# B&R Automation Studio project vibratorControlWithCurrentController (part 3)

#### brdkEM.c - Represents an equipment module.
```c
#include <brdkEM_func.h>

void brdkEM(struct brdkEM* this) {

	brdkEM_typ* parent;
	wakeMU(this->internal.muList.idx,(unsigned long)this);
	parent = getEm(this->internal.muList.parentIdx);

	/* if enabled command state completet can be set by settings the sub state to SC (65000) */
	if(this->setup.useSubstateSC) this->internal.cmdSC = this->substate == SC ? true : this->cmd.sc;
	else this->internal.cmdSC = this->cmd.sc;

	/* update information about the last */

	switch(this->state) {

		case STATE_STOPPED:
			this->status.color = BLUE;
			lightTree(this,BLUE,RED);
			setSubStateText(this);
			observeChildrensState(this, 2, STATE_ABORTING, STATE_ABORTED);						/* check if a child is in STATE- ABORTING or ABORTED */
			observeParentState(this, parent, 2, STATE_RESETTING, STATE_ABORTING);					/* check if parent is in STATE- RESETTING */
			if(this->internal.findParent) findParent(this,parent,STATE_RESETTING,11,STATE_IDLE,STATE_STARTING,STATE_EXECUTE,STATE_HOLDING,STATE_HELD,STATE_UNHOLDING,STATE_SUSPENDING,STATE_SUSPENDED,STATE_UNSUSPENDING,STATE_COMPLETING,STATE_COMPLETE);
			checkCommands(this, parent, 3, STATE_RESETTING, STATE_ABORTING, STATE_DEACTIVATING);		/* check commands reset, abort, not activate */
			setChildrenMode(this);
			if(this->mode == MODE_UNDEFINED) this->mode = MODE_PRODUCING;
			this->status.level = parent != NULL ? parent->status.level+1  : 0;	/* sets the hierarchy level */
			break;

		case STATE_RESETTING:
			this->status.color = WHITE;
			lightTree(this,BLUE,WHITE);
			setSubStateText(this);
			checkChildren(this, STATE_IDLE); 													/* CHECK IF ALL CHILDREN ARE IN STATE_IDLE */
			observeChildrensState(this, 3, STATE_ABORTING, STATE_ABORTED, STATE_STOPPING);		/* CHECK IF ONE CHILD IS IN STATE_ABORTING OR STATE_ABORTED */
			observeParentState(this,parent, 2, STATE_STOPPING,STATE_ABORTING);							/* checks if parent is in STATE- STOPPING or ABORTING */
			checkCommands(this, parent, 2, STATE_STOPPING, STATE_ABORTING);								/* check commands stop and abort */
			break;

		case STATE_IDLE:
			this->status.color = BLUE;
			lightTree(this,BLUE,WHITE);
			setSubStateText(this);
			observeChildrensState(this, 4, STATE_ABORTING, STATE_ABORTED, STATE_STOPPING, STATE_STOPPED);		/* check child state */
			observeParentState(this, parent, 3,STATE_STARTING,STATE_STOPPING,STATE_ABORTING);						/* CHECK STATE OF THE PARENT AND MAYBE FOLLOW */
			if(this->internal.findParent) findParent(this,parent,STATE_STARTING,9,STATE_EXECUTE,STATE_HOLDING,STATE_HELD,STATE_UNHOLDING,STATE_SUSPENDING,STATE_SUSPENDED,STATE_UNSUSPENDING,STATE_COMPLETING,STATE_COMPLETE);
			checkCommands(this, parent, 3, STATE_STOPPING, STATE_ABORTING, STATE_STARTING);								/* check commands stop, abort, start */
			break;

		case STATE_STARTING:
			this->status.color = WHITE;
			lightTree(this,flashColor(this,GREEN),WHITE);
			setSubStateText(this);
			checkChildren(this, STATE_EXECUTE); 															/* SUBSTATE MUST BE IN SC - CHECK IF ALL CHILDREN ARE IN STATE_EXECUTE */
			observeChildrensState(this, 4, STATE_ABORTING, STATE_ABORTED, STATE_STOPPING, STATE_STOPPED);	/* CHECK IF ONE CHILD IS IN STATE */
			observeParentState(this, parent,2,STATE_STOPPING,STATE_ABORTING); 										/* CHECK STATE OF THE PARENT AND MAYBE FOLLOW */
			checkCommands(this, parent, 2, STATE_STOPPING, STATE_ABORTING);											/* check commands stop, abort */
			break;

		case STATE_EXECUTE:
			this->status.color = GREEN;
			lightTree(this,GREEN,WHITE);
			setSubStateText(this);
			observeChildrensState(this, 8, STATE_ABORTING, STATE_ABORTED, STATE_STOPPING, STATE_STOPPED, STATE_SUSPENDING, STATE_SUSPENDED, STATE_HOLDING, STATE_HELD);		/* CHECK IF ONE CHILD IS IN STATE */
			observeParentState(this,parent,5,STATE_HOLDING,STATE_SUSPENDING,STATE_COMPLETING,STATE_STOPPING,STATE_ABORTING); /* CHECK STATE OF THE PARENT AND MAYBE FOLLOW */
			if(this->internal.findParent) findParent(this,parent,STATE_EXECUTE,7,STATE_HOLDING,STATE_HELD,STATE_SUSPENDING,STATE_SUSPENDED,STATE_COMPLETING,STATE_COMPLETE);
			checkCommands(this, parent, 5, STATE_STOPPING, STATE_ABORTING, STATE_HOLDING, STATE_SUSPENDING, STATE_COMPLETING);		/* check commands stop, abort, hold, suspend, complete */
			break;

		case STATE_HOLDING:
			this->status.color = WHITE;
			lightTree(this,flashColor(this,RED),WHITE);
			setSubStateText(this);
			checkChildren(this, STATE_HELD); 											/* SUBSTATE MUST BE IN SC - CHECK IF ALL CHILDREN ARE IN STATE_EXECUTE */
			observeChildrensState(this, 2, STATE_ABORTING, STATE_ABORTED);				/* CHECK IF ONE CHILD IS IN STATE */
			observeParentState(this,parent,2,STATE_STOPPING,STATE_ABORTING); 					/* CHECK STATE OF THE PARENT AND MAYBE FOLLOW */
			checkCommands(this, parent, 2, STATE_STOPPING, STATE_ABORTING);						/* check commands stop, abort */
			break;

		case STATE_HELD:
			this->status.color = RED;
			lightTree(this,flashColor(this,RED),WHITE);
			setSubStateText(this);
			observeChildrensState(this, 2, STATE_ABORTING, STATE_ABORTED);					/* CHECK IF ONE CHILD IS IN STATE */
			observeParentState(this,parent,3,STATE_UNHOLDING,STATE_STOPPING,STATE_ABORTING); 	/* CHECK STATE OF THE PARENT AND MAYBE FOLLOW */
			if(this->internal.findParent) findParent(this,parent,STATE_UNHOLDING,6,STATE_EXECUTE,STATE_SUSPENDING,STATE_SUSPENDED,STATE_UNSUSPENDING,STATE_COMPLETING,STATE_COMPLETE);
			checkCommands(this, parent, 3, STATE_STOPPING, STATE_ABORTING, STATE_UNHOLDING);		/* check commands stop, abort, start */
			break;

		case STATE_UNHOLDING:
			this->status.color = WHITE;
			lightTree(this,RED,GREEN);
			setSubStateText(this);
			checkChildren(this, STATE_EXECUTE); 											/* SUBSTATE MUST BE IN SC - CHECK IF ALL CHILDREN ARE IN STATE_EXECUTE */
			observeChildrensState(this, 2, STATE_ABORTING, STATE_ABORTED);					/* CHECK IF ONE CHILD IS IN STATE */
			observeParentState(this,parent,2,STATE_STOPPING,STATE_ABORTING); 						/* CHECK STATE OF THE PARENT AND MAYBE FOLLOW */
			checkCommands(this, parent, 2, STATE_STOPPING, STATE_ABORTING);							/* check commands stop, abort */
			break;

		case STATE_SUSPENDING:
			this->status.color = WHITE;
			lightTree(this,ORANGE,WHITE);
			setSubStateText(this);
			checkChildren(this, STATE_SUSPENDED); 											/* SUBSTATE MUST BE IN SC - CHECK IF ALL CHILDREN ARE IN STATE_EXECUTE */
			observeChildrensState(this, 2, STATE_ABORTING, STATE_ABORTED);					/* CHECK IF ONE CHILD IS IN STATE */
			observeParentState(this,parent,2,STATE_STOPPING,STATE_ABORTING); 						/* CHECK STATE OF THE PARENT AND MAYBE FOLLOW */
			checkCommands(this, parent, 2, STATE_STOPPING, STATE_ABORTING);							/* check commands stop, abort */
			break;

		case STATE_SUSPENDED:
			this->status.color = ORANGE;
			lightTree(this,ORANGE,WHITE);
			setSubStateText(this);
			observeChildrensState(this, 2, STATE_ABORTING, STATE_ABORTED);					/* CHECK IF ONE CHILD IS IN STATE */
			observeParentState(this,parent,3,STATE_UNSUSPENDING,STATE_STOPPING,STATE_ABORTING); 	/* CHECK STATE OF THE PARENT AND MAYBE FOLLOW */
			if(this->internal.findParent) findParent(this,parent,STATE_UNSUSPENDING,6,STATE_EXECUTE,STATE_HOLDING,STATE_HELD,STATE_UNHOLDING,STATE_COMPLETING,STATE_COMPLETE);
			checkCommands(this, parent, 3, STATE_STOPPING, STATE_ABORTING, STATE_UNSUSPENDING);		/* check commands stop, abort, start */
			break;

		case STATE_UNSUSPENDING:
			this->status.color = WHITE;
			lightTree(this,ORANGE,GREEN);
			setSubStateText(this);
			checkChildren(this, STATE_EXECUTE); 											/* SUBSTATE MUST BE IN SC - CHECK IF ALL CHILDREN ARE IN STATE_EXECUTE */
			observeChildrensState(this, 2, STATE_ABORTING, STATE_ABORTED);					/* CHECK IF ONE CHILD IS IN STATE */
			observeParentState(this,parent,2,STATE_STOPPING,STATE_ABORTING); 						/* CHECK STATE OF THE PARENT AND MAYBE FOLLOW */
			checkCommands(this, parent, 2, STATE_STOPPING, STATE_ABORTING);							/* check commands stop, abort */
			break;

		case STATE_COMPLETING:
			this->status.color = WHITE;
			lightTree(this,GREEN,BLUE);
			setSubStateText(this);
			checkChildren(this, STATE_COMPLETE); 											/* SUBSTATE MUST BE IN SC - CHECK IF ALL CHILDREN ARE IN STATE_EXECUTE */
			observeChildrensState(this, 2, STATE_ABORTING, STATE_ABORTED);					/* CHECK IF ONE CHILD IS IN STATE */
			observeParentState(this,parent,2,STATE_STOPPING,STATE_ABORTING); 						/* CHECK STATE OF THE PARENT AND MAYBE FOLLOW */
			checkCommands(this, parent, 2, STATE_STOPPING, STATE_ABORTING);							/* check commands stop, abort */
			break;

		case STATE_COMPLETE:
			this->status.color = BLUE;
			lightTree(this,flashColor(this,BLUE),WHITE);
			setSubStateText(this);
			observeChildrensState(this, 2, STATE_ABORTING, STATE_ABORTED);					/* CHECK IF ONE CHILD IS IN STATE */
			observeParentState(this,parent,3,STATE_RESETTING,STATE_STOPPING,STATE_ABORTING); 		/* CHECK STATE OF THE PARENT AND MAYBE FOLLOW */
			if(this->internal.findParent) findParent(this,parent,STATE_RESETTING,10,STATE_IDLE,STATE_STARTING,STATE_EXECUTE,STATE_HOLDING,STATE_HELD,STATE_UNHOLDING,STATE_SUSPENDING,STATE_SUSPENDED,STATE_UNSUSPENDING,STATE_COMPLETING);
			checkCommands(this, parent, 3, STATE_STOPPING, STATE_ABORTING, STATE_RESETTING);		/* check commands stop, abort, reset */
			break;

		case STATE_ABORTING:
			this->status.color = WHITE;
			lightTree(this,RED,WHITE);
			setSubStateText(this);
			checkChildren(this, STATE_ABORTED);
			break;

		case STATE_ABORTED:
			this->status.color = RED;
			lightTree(this,RED,WHITE);
			setSubStateText(this);
			observeParentState(this,parent,1,STATE_CLEARING); 										/* CHECK STATE OF THE PARENT AND MAYBE FOLLOW */
			checkCommands(this, parent, 2, STATE_CLEARING, STATE_DEACTIVATING);						/* check commands clar, not activate */
			break;

		case STATE_CLEARING:
			this->status.color = WHITE;
			lightTree(this,RED,flashColor(this,BLUE));
			setSubStateText(this);
			checkChildren(this, STATE_STOPPED); 										/* SUBSTATE MUST BE IN SC - CHECK IF ALL CHILDREN ARE IN STATE_EXECUTE */
			observeChildrensState(this, 2, STATE_ABORTING, STATE_ABORTED);				/* CHECK IF ONE CHILD IS IN STATE */
			observeParentState(this,parent,2,STATE_STOPPING,STATE_ABORTING); 			/* CHECK STATE OF THE PARENT AND MAYBE FOLLOW */
			break;

		case STATE_STOPPING:
			this->status.color = WHITE;
			lightTree(this,GREEN,BLUE);
			setSubStateText(this);
			checkChildren(this, STATE_STOPPED); 									/* SUBSTATE MUST BE IN SC - CHECK IF ALL CHILDREN ARE IN STATE_EXECUTE */
			observeChildrensState(this, 2, STATE_ABORTING, STATE_ABORTED);			/* CHECK IF ONE CHILD IS IN STATE */
			observeParentState(this,parent,1,STATE_ABORTING); 								/* CHECK STATE OF THE PARENT AND MAYBE FOLLOW */
			checkCommands(this, parent, 2, STATE_ABORTING, STATE_DEACTIVATING);								/* check commands abort */
			break;

		case STATE_DEACTIVATING:
			this->status.color = WHITE;
			lightTree(this,flashColor(this,GREY),WHITE);
			setSubStateText(this);
			this->mode = MODE_UNDEFINED;
			this->internal.initSubstate = 0;
			if(this->internal.cmdSC) {
				UnregisterChild(this, parent);
				this->state = STATE_DEACTIVATED;
			}
			break;

		case STATE_ACTIVATING:
			this->status.color = WHITE;
			lightTree(this,flashColor(this,GREY),BLUE);
			setSubStateText(this);
			if(this->internal.cmdSC) {
				if(parent != NULL) {
					switch(parent->state) {

						case STATE_STOPPED:
							if(this->mode == MODE_UNDEFINED && this->setup.reactTo == BRDK_EM_REACT_TO_NONE) this->mode = MODE_PRODUCING;
							else this->mode = parent->mode;
							this->state = STATE_STOPPED;
							break;

						case STATE_DEACTIVATED:
							brdkStrCpy((unsigned long)this->status.substate,(unsigned long)"waiting for parent to be activated");
							break;

						default:
							brdkStrCpy((unsigned long)this->status.substate,(unsigned long)"waiting for parent to be in STATE_STOPPED");
							break;

					}
				}
				else {
					if(this->mode == MODE_UNDEFINED) this->mode = MODE_PRODUCING;
					this->state = STATE_STOPPED;
				}
			}
			break;

		case STATE_DEACTIVATED:
			brdkStrCpy((unsigned long)this->status.state,(unsigned long)brdkEMStateToA(this->state));
			this->status.color = GREY;
			lightTree(this,GREY,WHITE);
			setSubStateText(this);
			if(this->status.mode[0] == 0) brdkStrCpy((unsigned long)this->status.mode,brdkEMModeToA(this->mode));
			if(this->status.cycleTime == 0) this->status.cycleTime = getCycleTime();								/* get the modules cycle time */
			brdkEMInitialize(this,parent);
			checkCommands(this, parent, 1, STATE_ACTIVATING);
			break;
	}

	/* mode change */
	if(this->mode != this->internal.old.mode) {
		if(this->state == STATE_STOPPED || this->state == STATE_ACTIVATING || this->state == STATE_DEACTIVATING || this->state == STATE_DEACTIVATED) {
			/* save last state for log */
			if(this->setup.lastActivated) {
				brdkStrMemMove((unsigned long)this->status.last[1],(unsigned long)this->status.last[0], sizeof(this->status.last[0])*BRDK_MU_MAX_LAST_SIZE);
				brdkStrCpy((unsigned long)this->status.last[0], brdkEMModeToA(this->internal.old.mode));
				brdkStrCat((unsigned long)this->status.last[0], (unsigned long)"-->");
				brdkStrCat((unsigned long)this->status.last[0], brdkEMModeToA(this->mode));
			}
			this->internal.old.mode = this->mode;
			brdkStrCpy((unsigned long)this->status.mode,brdkEMModeToA(this->mode));
		}
		else { /* avoid mode being change in other states than STATE_STOPPED */
			this->status.unvalidatedMode = true;
			this->mode = this->internal.old.mode;
		}
	}

	this->status.time += this->status.cycleTime/1000;

	/* state change */
	if(this->state != this->internal.old.state || this->substate != this->internal.old.substate) {
		/* save last state for log */
		if(this->setup.lastActivated) {
			brdkStrMemMove((unsigned long)this->status.last[1],(unsigned long)this->status.last[0], sizeof(this->status.last[0])*BRDK_MU_MAX_LAST_SIZE);
			brdkStrCpy((unsigned long)this->status.last[0],(unsigned long)this->status.state);
			brdkStrCat((unsigned long)this->status.last[0],(unsigned long)": ");
			if(this->state != this->internal.old.state) brdkStrAppendUdintToA(this->substate,(unsigned long)this->status.last[0],BRDK_STR_CONVERT_DECIMAL,-1);
			else brdkStrAppendUdintToA(this->internal.old.substate,(unsigned long)this->status.last[0],BRDK_STR_CONVERT_DECIMAL,-1);
			brdkStrCat((unsigned long)this->status.last[0],(unsigned long)": ");
			brdkStrAppendUdintToA(this->status.time,(unsigned long)this->status.last[0],BRDK_STR_CONVERT_DECIMAL,-1);
			brdkStrCat((unsigned long)this->status.last[0],(unsigned long)"ms");
		}
		brdkStrCpy((unsigned long)this->status.state,(unsigned long)brdkEMStateToA(this->state));
		if(this->state != this->internal.old.state) {
			/* log who interrupted the module */
			if(this->internal.pInterrupter != 0 && this->status.interruptedBy.name[0] == 0) {
				brdkStrCpy((unsigned long)this->status.interruptedBy.name,(unsigned long)((brdkEM_typ*)this->internal.pInterrupter)->status.name);
				if(this->internal.pInterrupter != (unsigned long)this) {
					this->status.interruptedBy.state = ((brdkEM_typ*)this->internal.pInterrupter)->status.interruptedBy.state;
					this->status.interruptedBy.substate = ((brdkEM_typ*)this->internal.pInterrupter)->status.interruptedBy.substate;
				}
				else {
					this->status.interruptedBy.state = ((brdkEM_typ*)this->internal.pInterrupter)->internal.old.state;
					this->status.interruptedBy.substate = ((brdkEM_typ*)this->internal.pInterrupter)->internal.old.substate;
				}
				if(this->state == STATE_ABORTING || this->state == STATE_STOPPING) {
					if(this->setup.lastActivated) {
						brdkStrMemMove((unsigned long)this->status.last[1],(unsigned long)this->status.last[0], sizeof(this->status.last[0])*BRDK_MU_MAX_LAST_SIZE);
						if(this->state == STATE_ABORTING) brdkStrCpy((unsigned long)this->status.last[0],(unsigned long)"Aborted by: ");
						else brdkStrCpy((unsigned long)this->status.last[0],(unsigned long)"Stopped by: ");
						brdkStrCat((unsigned long)this->status.last[0],(unsigned long)this->status.interruptedBy.name);
						brdkStrCat((unsigned long)this->status.last[0],(unsigned long)": ");
						brdkStrCat((unsigned long)this->status.last[0],brdkEMStateToA(this->status.interruptedBy.state));
						brdkStrCat((unsigned long)this->status.last[0],(unsigned long)": ");
						brdkStrAppendUdintToA(this->status.interruptedBy.substate,(unsigned long)this->status.last[0],BRDK_STR_CONVERT_DECIMAL,-1);
					}
				}
			}
			this->internal.cmdSC = this->cmd.sc = this->cmd.start = this->cmd.reset = this->cmd.abort = this->cmd.stop = this->cmd.clear = this->cmd.hold = this->cmd.complete = this->cmd.suspend = false; /* reset commands when the state changes */
			this->substate = 0;	/* reset substate by a state change */
			this->status.time = 0;
			this->status.unvalidatedMode = false;
		}
		this->status.substate[0] = this->description[0] = 0;
		this->internal.old.state = this->state;
		this->internal.old.substate = this->substate;

	}

	/* update parent info */
	if(parent != NULL) {
		this->status.parent.state = parent->state;
		this->status.parent.substate = parent->substate;
		this->status.parent.sleeping = parent->status.sleeping;
		this->status.parent.mode = parent->mode;
		this->status.parent.sc = parent->cmd.sc;
		if(parent->setup.skipStopSC) this->setup.skipStopSC = true; /* check if skipStopSC is set in parent module */
	}

	/* reactTo has changed */
	if(this->internal.old.reactTo != this->setup.reactTo) {
		if(this->setup.reactTo == BRDK_EM_REACT_TO_ALL) {
			if(parent != NULL) this->internal.findParent = true;
		}
		this->internal.old.reactTo = this->setup.reactTo;
	}

	/* update siblings info */
	updateSiblingInfo(&this->internal.muList.siblingIdx, &this->status.sibling[0]);

	/* save the restore information */
	if(this->setup.restore.activate) {
		if(this->setup.restore.pRestoreStruct != 0) {
			this->setup.restore.pRestoreStruct->mode = this->mode;
			this->setup.restore.pRestoreStruct->state = this->state;
			this->setup.restore.pRestoreStruct->substate = this->substate;
			this->setup.restore.pRestoreStruct->sc = this->internal.cmdSC;
		}
	}
}
```

#### brdkEMSleep.c - Put an equipment module to sleep. It's pointer is added to a sleeping module list where it can be found again by brdkEMWake().
```c
#include <brdkMU_func.h>

signed long brdkEMSleep(unsigned long pEM) {
	brdkEM_typ* this;
	if(pEM != 0) {
		this = (brdkEM_typ*)pEM;
		this->status.sleeping = true;
		if(this->setup.lastActivated) {
			brdkStrMemMove((unsigned long)this->status.last[1],(unsigned long)this->status.last[0], sizeof(this->status.last[0])*BRDK_MU_MAX_LAST_SIZE);
			brdkStrCpy((unsigned long)this->status.last[0],(unsigned long)"module put to sleep");
		}
		return sleepMU(this->internal.muList.idx, pEM);
	}
	return -1;
}
```

#### brdkEMModeToA.c - Converts an equipment module mode constant to a string representation.
```c
#include <brdkEM_func.h>

unsigned long brdkEMModeToA(signed long mode) {
	unsigned long pStr;
	switch(mode) {
		case MODE_UNDEFINED: 	pStr = (unsigned long)&"MODE_UNDEFINED"; 	break;	/* 0 */
		case MODE_PRODUCING: 	pStr = (unsigned long)&"MODE_PRODUCING"; 	break;	/* 1 */
		case MODE_MAINTENANCE: 	pStr = (unsigned long)&"MODE_MAINTENANCE"; 	break;	/* 2 */
		case MODE_MANUAL: 		pStr = (unsigned long)&"MODE_MANUAL"; 		break;	/* 3 */
		case MODE_CLEAN: 		pStr = (unsigned long)&"MODE_CLEAN"; 		break;	/* 16 */
		case MODE_JOG: 			pStr = (unsigned long)&"MODE_JOG"; 			break;	/* 17 */
		case MODE_CIP: 			pStr = (unsigned long)&"MODE_CIP"; 			break;	/* 18 */
		case MODE_CALIBRATING: 	pStr = (unsigned long)&"MODE_CALIBRATING"; 	break;	/* 19 */
		default: pStr = (unsigned long)&""; 	break;
	}
	return pStr;
}
```

#### brdkEM_func.c - Internal functions for brdkEM.
```c
#include <brdkEM_func.h>

static unsigned char semCreator = false;
SemCreate_typ SemCreateMUList;

/* initialize the equipment module */
void brdkEMInitialize(brdkEM_typ* this, brdkEM_typ* parent) {
	int i;
	brdk_mu_setup_module_typ module;

	switch(this->internal.initSubstate) {

		case 0:
			if(this->setup.name[0] == 0) ST_name(0,(char*)&this->setup.name,(unsigned char)0); 														/* set module name to task name if not set*/
			brdkStrCpy((unsigned long)this->status.name,(unsigned long)this->setup.name);
			if(this->setup.nameIdx > -1) brdkStrAppendUdintToA(this->setup.nameIdx,(unsigned long)&this->status.name, BRDK_STR_CONVERT_DECIMAL,-1);	/* add index to task name */
			this->internal.muList.parentIdx = -1;
			for(i=0; i<= BRDK_EM_MAX_CHILDREN; i++) this->internal.muList.childrenIdx[i] = -1;
			for(i=0; i<= BRDK_MU_MAX_SIBLINGS; i++) this->internal.muList.siblingIdx[i] = -1;
			if(!semCreator) {
				brdkStrCpy((unsigned long)this->status.substate,(unsigned long)"creating global semaphore");
				semCreator = true;
				this->internal.initSubstate = 10;
			}
			else this->internal.initSubstate = 20;
			break;

		case 10:
			SemCreateMUList.enable = true;
			SemCreateMUList.initCount = 0;
			SemCreateMUList.maxCount = 1;
			SemCreate(&SemCreateMUList);
			if(SemCreateMUList.status != ERR_OK) brdkStrCpy((unsigned long)this->status.substate,(unsigned long)"creating global semaphore");
			else {
				SemRelease(SemCreateMUList.ident);
				this->internal.muList.idx = addToMUList((unsigned long)this,0);
				if(this->internal.muList.idx != -1) {
					emListReady = true;
					this->internal.initSubstate = !this->setup.parent.name[0] ? 40 : 30;	/* check if the module has a parent name assigned */
				}
				else {
					brdkStrCpy((unsigned long)this->status.substate,(unsigned long)"em list full. Expand BRDK_EM_MAX_EMS.");
					this->internal.initSubstate = 200;
				}
			}
			break;

		case 20:	/* add module to em list */
			if(!emListReady) brdkStrCpy((unsigned long)this->status.substate,(unsigned long)"waiting for em list to be ready");
			else {
				brdkStrCpy((unsigned long)module.name,(unsigned long)this->setup.name);
				module.index = this->setup.nameIdx;
				this->internal.muList.idx = getMUIndex((unsigned long)this, &module);
				if(this->internal.muList.idx != -1) {
					if(moduleSleeping(this->internal.muList.idx)) {
						wakeMU(this->internal.muList.idx,(unsigned long)this);
						if(this->setup.lastActivated) {
							brdkStrMemMove((unsigned long)this->status.last[1],(unsigned long)this->status.last[0], sizeof(this->status.last[0])*BRDK_MU_MAX_LAST_SIZE);
							brdkStrCpy((unsigned long)this->status.last[0],(unsigned long)"module awake");
						}
						this->internal.initSubstate = 65000;
					}
					else {	/* module name already exists in the list */
						brdkStrCpy((unsigned long)this->status.substate,(unsigned long)"module name ");
						brdkStrCat((unsigned long)this->status.substate,(unsigned long)module.name);
						brdkStrCat((unsigned long)this->status.substate,(unsigned long)" already used. Rename module.");
						this->internal.muList.idx = -1;
						this->internal.initSubstate = 100;
					}
				}
				else {
					if(SemAcquire(SemCreateMUList.ident) != ERR_OK) brdkStrCpy((unsigned long)this->status.substate,(unsigned long)"waiting global semaphore to be free");
					else {
						this->internal.muList.idx = addToMUList((unsigned long)this,0);
						SemRelease(SemCreateMUList.ident);
						brdkStrCpy((unsigned long)this->status.substate,(unsigned long)"module added em list");
						if(this->internal.muList.idx != -1) this->internal.initSubstate = !this->setup.parent.name[0] ? 40 : 30;	/* check if the module has a parent name assigned */
						else {
							brdkStrCpy((unsigned long)this->status.substate,(unsigned long)"em list full. Expand BRDK_EM_MAX_EMS.");
							this->internal.initSubstate = 200;
						}
					}
				}
			}
			break;

		case 30:	/* find parent */
			this->internal.muList.parentIdx = getMUIndex((unsigned long)this, &this->setup.parent);
			if(this->internal.muList.parentIdx == -1) brdkStrCpy((unsigned long)this->status.substate,(unsigned long)"parent not found");
			else this->internal.initSubstate = 40;
			break;

		case 40:	/* find siblings */
			for(i=0; i<= BRDK_MU_MAX_SIBLINGS; i++) {
				if(this->setup.sibling[i].name[0] != 0) {
					this->internal.muList.siblingIdx[i] = getMUIndex((unsigned long)this, &this->setup.sibling[i]);
					if(this->internal.muList.siblingIdx[i] == -1) {
						brdkStrCpy((unsigned long)this->status.substate,(unsigned long)"sibling: ");
						brdkStrCat((unsigned long)this->status.substate,(unsigned long)this->setup.sibling[i].name);
						brdkStrCat((unsigned long)this->status.substate,(unsigned long)" not found");
						break;
					}
				}
			}
			if(i>=BRDK_MU_MAX_SIBLINGS) {
				this->status.substate[0] = 0;	/* reset status text */
				this->internal.initSubstate = this->internal.SemCreate_0.ident == 0 ? 50 : 60;
			}
			break;

		case 50:
			this->internal.SemCreate_0.enable = true;
			this->internal.SemCreate_0.initCount = 0;
			this->internal.SemCreate_0.maxCount = 1;
			SemCreate(&this->internal.SemCreate_0);
			switch(this->internal.SemCreate_0.status) {

				case 0:	/* ERR_OK */
					SemRelease(this->internal.SemCreate_0.ident);		/* release the semaphore so it's ready */
					this->internal.initSubstate = 60;
					break;

				case 65535:	/* ERR_FUB_BUSY */
					break;

				default:
					brdkStrCpy((unsigned long)this->status.substate,(unsigned long)"error creating the semaphore");
					break;

			}
			break;

		case 60:
			brdkStrCpy((unsigned long)this->status.substate,(unsigned long)"register child to parent");
			if(RegisterChild(this, parent) == 0) {
				this->internal.initSubstate = 65000;				/* add child to parent's children list */
				if(this->substate == 0) this->substate = 65000;		/* if substate is still 0 it's auto set to SC */
			}
			break;

		case 100: /* error module name already used. Check if anme is being changed */
			if(brdkStrCmp((unsigned long)module.name,(unsigned long)this->setup.name) != 0) {
				this->internal.initSubstate = 20;
			}
			break;

	}
}

/* traverse and find the real interrupter */
unsigned long findInterrupter(unsigned long pEM) {
	if(((brdkEM_typ*)pEM)->internal.pInterrupter != pEM) return findInterrupter(((brdkEM_typ*)pEM)->internal.pInterrupter);
	return pEM;
}

/* flash functionality */
brdk_em_color_typ flashColor(brdkEM_typ* this, brdk_em_color_typ color) {
	if(this->internal.flashTime >= BRDK_EM_FLASH_TIME*2) this->internal.flashTime = 0;
	else this->internal.flashTime += this->status.cycleTime/1000;
	return this->internal.flashTime >= BRDK_EM_FLASH_TIME ? color : WHITE;
}

/* light tree functionality */
void lightTree(brdkEM_typ* this, brdk_em_color_typ color1, brdk_em_color_typ color2) {
	this->status.lightTree.red 		= color1 == RED || color2 == RED;
	this->status.lightTree.yellow 	= color1 == ORANGE || color2 == ORANGE;
	this->status.lightTree.blue 	= color1 == BLUE || color2 == BLUE;
	this->status.lightTree.green 	= color1 == GREEN || color2 == GREEN;
}

/* set default sub state text if not set in program */
void setSubStateText(brdkEM_typ* this) {
	if(this->status.substate[0] == 0) {
		if(this->description[0] == 0) {
			if(this->substate == 0) brdkStrCpy((unsigned long)this->status.substate,(unsigned long)"0: waiting for state change (SC)");
			else if(this->internal.cmdSC) {
				switch(this->state) {
					case STATE_DEACTIVATED: brdkStrCpy((unsigned long)this->status.substate, (unsigned long)"SC: waiting for activate command"); break;
					case STATE_STOPPED: case STATE_COMPLETE: brdkStrCpy((unsigned long)this->status.substate, (unsigned long)"SC: waiting for reset command"); break;
					case STATE_IDLE: case STATE_SUSPENDED: case STATE_HELD:	brdkStrCpy((unsigned long)this->status.substate, (unsigned long)"SC: waiting for start command"); break;
					case STATE_ABORTED: brdkStrCpy((unsigned long)this->status.substate, (unsigned long)"SC: waiting for clear command"); break;
					default: break;
				}
			}
		}
		else {
			brdkStrUdintToA(this->substate,(unsigned long)&this->status.substate,BRDK_STR_CONVERT_DECIMAL);
			brdkStrCat((unsigned long)this->status.substate, (unsigned long)": ");
			brdkStrCat((unsigned long)this->status.substate, (unsigned long)this->description);
		}
	}
}

/* if the parent mode is changed we also changes it for alle the children */
void setChildrenMode(brdkEM_typ* this) {
	int i;
	for(i=0; i <= BRDK_EM_MAX_CHILDREN; i++) {
		brdkEM_typ* child = getEm(this->internal.muList.childrenIdx[i]);
		if(child != NULL) {
			if(this->setup.reactTo == BRDK_EM_REACT_TO_NONE) child->mode = child->mode;
			else child->mode = this->mode;
		}
		else break;
	}
}

/* CHECKS IF ALL THE CHILDREN IS IN STATE */
void checkChildren(brdkEM_typ* this, brdk_em_states_typ STATE) {
	brdkEM_typ* parent;
	brdkEM_typ* child;
	if(this->internal.cmdSC) {
		int i = 0, j;
		this->status.waitingFor.name[0] = 0;
		this->status.waitingFor.substate[0] = 0;
		while(i < this->status.childCount) {
			child = getEm(this->internal.muList.childrenIdx[i]);
			if(child != NULL) {
				j = i;
				if(child->state == STATE_ACTIVATING || child->state == STATE_DEACTIVATED || child->state == STATE_DEACTIVATING) i++;
				else {
					switch(child->setup.reactTo) {

						case BRDK_EM_REACT_TO_ALL:
							if(child->state == STATE) i++;
							break;

						case BRDK_EM_REACT_TO_ABORT_AND_STOP:
							if(STATE == STATE_ABORTED || STATE == STATE_STOPPED) {
								if(child->state == STATE) i++;
							}
							else i++;
							break;

						case BRDK_EM_REACT_TO_ABORT_ONLY:
							if(STATE == STATE_ABORTED) {
								if(child->state == STATE) i++;
							}
							else i++;
							break;

						case BRDK_EM_REACT_TO_STOP_ONLY:
							if(STATE == STATE_STOPPED) {
								if(child->state == STATE) i++;
							}
							else i++;
							break;

						case BRDK_EM_REACT_TO_NONE: case BRDK_EM_LISTEN_TO_ABORT_AND_STOP: case BRDK_EM_LISTEN_TO_ABORT_ONLY: case BRDK_EM_LISTEN_TO_STOP_ONLY:
							i++;
							break;

					}
				}
				if(j == i) {	/* index not increased */
					if(!this->status.waitingFor.name[0]) {
						if(child->status.waitingFor.name[0] != 0) {	/* check to see if a child is also waiting for someone */
							brdkStrCpy((unsigned long)this->status.waitingFor.name,(unsigned long)child->status.waitingFor.name);
							brdkStrCpy((unsigned long)this->status.waitingFor.substate,(unsigned long)child->status.waitingFor.substate);
						}
						else {
							brdkStrCpy((unsigned long)this->status.waitingFor.name,(unsigned long)child->setup.name);
							brdkStrCpy((unsigned long)this->status.waitingFor.substate,(unsigned long)child->status.substate);
							brdkStrCpy((unsigned long)this->status.substate, (unsigned long)"SC: waiting for ");
							brdkStrCat((unsigned long)this->status.substate, (unsigned long)this->status.waitingFor.name);
							if(brdkStrLen((unsigned long)this->status.waitingFor.substate) + 2 >= BRDK_MU_MAX_DESCRIPTION_STRING - brdkStrLen((unsigned long)this->status.substate)) { /* skip if too long */
								brdkStrCat((unsigned long)this->status.substate, (unsigned long)", ");
								brdkStrCat((unsigned long)this->status.substate, (unsigned long)this->status.waitingFor.substate);
							}
						}
					}
					break;
				}
			}
			else break;
		}
		if(parentStateOK(this)) {
			if(i==this->status.childCount) {
				if(this->state == STATE_RESETTING || this->state == STATE_CLEARING) {	/* clear interrupted by data */
					brdkStrMemSet((unsigned long)&this->status.interruptedBy,0,sizeof(this->status.interruptedBy));
					this->internal.pInterrupter = 0;
				}
				this->state = STATE;
			}
		}
		else {
			if(!this->status.waitingFor.name[0]) {
				parent = getEm(this->internal.muList.parentIdx);
				if(parent != NULL) {
					if(parent->state == STATE_DEACTIVATED || parent->state == STATE_DEACTIVATING) brdkStrCpy((unsigned long)this->status.substate, (unsigned long)"SC: parent is deactivated");
					else brdkStrCpy((unsigned long)this->status.substate, (unsigned long)"SC: waiting for parent");
					brdkStrCpy((unsigned long)this->status.waitingFor.name,(unsigned long)parent->setup.name);
					brdkStrCpy((unsigned long)this->status.waitingFor.substate,(unsigned long)parent->status.substate);
				}
			}
		}
	}
}

/* make sure eventual parent is also in same state before state change */
int parentStateOK(brdkEM_typ* this) {
	int status = false;
	brdkEM_typ* parent = getEm(this->internal.muList.parentIdx);
	if(parent != NULL) {
		switch(this->setup.reactTo) {
			case BRDK_EM_REACT_TO_ALL: 				status = (parent->state == this->state || this->internal.findParent); break;
			case BRDK_EM_REACT_TO_ABORT_AND_STOP: 	status = (this->state == STATE_ABORTING || this->state == STATE_STOPPING) ? (parent->state == this->state) : true; break;
			case BRDK_EM_REACT_TO_ABORT_ONLY:		status = (this->state == STATE_ABORTING) ? (parent->state == this->state) : true; break;
			case BRDK_EM_REACT_TO_STOP_ONLY:		status = (this->state == STATE_STOPPING) ? (parent->state == this->state) : true; break;
			case BRDK_EM_REACT_TO_NONE: case BRDK_EM_LISTEN_TO_ABORT_AND_STOP: case BRDK_EM_LISTEN_TO_ABORT_ONLY: case BRDK_EM_LISTEN_TO_STOP_ONLY:	status = true;
		}
	}
	else status = true;
	return status;
}

/* automatically take the module to it's parents state */
void findParent(brdkEM_typ* this, brdkEM_typ* parent, brdk_em_states_typ cmd, int numArgs, ...) {
	if(parent != NULL) {
		va_list list;
		int i;
		if(this->state == parent->state) this->internal.findParent = false;
		else {
			va_start(list, numArgs);
			for(i=0; i < numArgs; i++) {
				brdk_em_states_typ checkState = va_arg(list, brdk_em_states_typ);
				if(parent->state == checkState) {
					switch(cmd) {
						case STATE_RESETTING: this->cmd.reset = true; break;
						case STATE_STARTING: case STATE_UNHOLDING: case STATE_UNSUSPENDING: this->cmd.start = true; break;
						case STATE_EXECUTE:
							switch(checkState) {
								case STATE_HOLDING: case STATE_HELD: this->cmd.hold = true; break;
								case STATE_SUSPENDING: case STATE_SUSPENDED: this->cmd.suspend = true; break;
								case STATE_COMPLETING: case STATE_COMPLETE: this->cmd.complete = true; break;
								default: break;
							}
							break;
						default: break;
					}
				}
			}
		}
	}
}

/* observes if one of the children is in one of the states */
void observeChildrensState(brdkEM_typ* this, int numArgs, ...) {
	int i,j;
	brdkEM_typ* child;
	va_list list;																					/* define argument list variable */
	for(i=0; i <= BRDK_EM_MAX_CHILDREN; i++) {														/* check all children */
		child = getEm(this->internal.muList.childrenIdx[i]);
		if(child != NULL) {											/* */
			brdk_em_setup_react_typ reactTo = child->setup.reactTo;
			if(reactTo == BRDK_EM_REACT_TO_NONE || reactTo == BRDK_EM_REACT_TO_NONE || reactTo == BRDK_EM_LISTEN_TO_ABORT_AND_STOP || reactTo == BRDK_EM_LISTEN_TO_ABORT_ONLY || reactTo == BRDK_EM_LISTEN_TO_STOP_ONLY) this->state = this->state;
			else {
				va_start(list, numArgs);
				for(j=0; j < numArgs; j++) {
					brdk_em_states_typ child_state = va_arg(list, brdk_em_states_typ);
					if(child->state == child_state) {
						switch(child_state) {

							case STATE_ABORTING:
								if(reactTo == BRDK_EM_REACT_TO_ALL || reactTo == BRDK_EM_REACT_TO_ABORT_AND_STOP || reactTo == BRDK_EM_REACT_TO_ABORT_ONLY) {
									this->internal.pInterrupter = findInterrupter((unsigned long)child); /* save who went in aborted or aborting */

									this->state = STATE_ABORTING;
								}
								break;

							case STATE_STOPPING:
								if((this->internal.cmdSC || this->setup.skipStopSC) && (reactTo == BRDK_EM_REACT_TO_ALL || reactTo == BRDK_EM_REACT_TO_ABORT_AND_STOP || reactTo == BRDK_EM_REACT_TO_STOP_ONLY)) {
									this->internal.pInterrupter = findInterrupter((unsigned long)child); /* save who went in stopped or stopping */
									this->state = STATE_STOPPING;
								}
								break;

							case STATE_SUSPENDING:
								if(this->internal.cmdSC && reactTo == BRDK_EM_REACT_TO_ALL) {
									this->internal.pInterrupter = findInterrupter((unsigned long)child); /* save who went in suspending or suspended */
									this->state = STATE_SUSPENDING;
								}
								break;

							case STATE_HOLDING:
								if(this->internal.cmdSC && reactTo == BRDK_EM_REACT_TO_ALL) {
									this->internal.pInterrupter = findInterrupter((unsigned long)child); /* save who went in holding or held */
									this->state = STATE_HOLDING;
								}
								break;

							default:
								break;

						}
						va_end(list);
						break;
					}
				}
			}
		}
		else {
			va_end(list);
			break;
		}
	}
}

/* observes the parent state by the given states */
void observeParentState(brdkEM_typ* this, brdkEM_typ* parent, int numArgs, ...) {
	int i;
	brdk_em_setup_react_typ reactTo =  this->setup.reactTo;
	if(parent == NULL || reactTo == BRDK_EM_REACT_TO_NONE) this->state = this->state;
	else {
		va_list list;																									/* define argument list variable */
		va_start(list, numArgs);																						/* init list */
		for(i=0; i < numArgs; i++) if(parent->state==va_arg(list, brdk_em_states_typ)) {
			switch(parent->state) {

				case STATE_ABORTING:
					if(reactTo == BRDK_EM_REACT_TO_ALL || reactTo == BRDK_EM_REACT_TO_ABORT_AND_STOP || reactTo == BRDK_EM_REACT_TO_ABORT_ONLY || reactTo == BRDK_EM_LISTEN_TO_ABORT_AND_STOP || reactTo == BRDK_EM_LISTEN_TO_ABORT_ONLY) {
						this->state = parent->state; 	/* get next state item and check if it's equal to parent state. and then set chils state*/
						this->internal.pInterrupter = parent->internal.pInterrupter;
					}
					break;

				case STATE_STOPPING:
					if((this->internal.cmdSC || this->setup.skipStopSC) && (reactTo == BRDK_EM_REACT_TO_ALL || reactTo == BRDK_EM_REACT_TO_ABORT_AND_STOP || reactTo == BRDK_EM_REACT_TO_STOP_ONLY || reactTo == BRDK_EM_LISTEN_TO_STOP_ONLY)) {
 						this->state = parent->state; 	/* get next state item and check if it's equal to parent state. and then set chils state*/
						this->internal.pInterrupter = parent->internal.pInterrupter;
					}
					break;

				case STATE_CLEARING:
					if(this->internal.cmdSC && (reactTo == BRDK_EM_REACT_TO_ALL || reactTo == BRDK_EM_REACT_TO_ABORT_AND_STOP || reactTo == BRDK_EM_REACT_TO_ABORT_ONLY)) this->state = parent->state; 	/* get next state item and check if it's equal to parent state. and then set chils state*/
					break;

				default:
					if(this->internal.cmdSC && reactTo == BRDK_EM_REACT_TO_ALL) this->state = parent->state; 	/* get next state item and check if it's equal to parent state. and then set chils state*/
					break;

			}
		}
		va_end(list);
	}																													/* cleanup the system stack */
}

/* check for commands -> STATE_STOPPING means check for command stop... */
void checkCommands(brdkEM_typ* this, brdkEM_typ* parent, int numArgs, ...) {
	brdkEM_typ* child;
	int i,j;
	if(this->internal.cmdSC || this->cmd.abort || (this->cmd.stop && this->setup.skipStopSC)) {
		va_list list;																											/* define argument list variable */
		va_start(list, numArgs);																								/* init list */
		for(i=0; i < numArgs; i++) {
			switch(va_arg(list, brdk_em_states_typ)) {

				case STATE_STOPPING:
					if(this->cmd.stop) {
						i = numArgs;
						this->internal.pInterrupter = (unsigned long)this; /* module interrupted itself */
						this->state = STATE_STOPPING;
					}
					break;

				case STATE_RESETTING:
					if(this->cmd.reset) {
						i = numArgs;
						this->state = STATE_RESETTING;
					}
					break;

				case STATE_CLEARING:
					if(this->cmd.clear) {
						this->state = STATE_CLEARING;
					}
					break;

				case STATE_STARTING:
					if(this->cmd.start) {
						i = numArgs;
						this->state = STATE_STARTING;
					}
					break;

				case STATE_HOLDING:
					if(this->cmd.hold) {
						i = numArgs;
						this->internal.pInterrupter = (unsigned long)this; /* module interrupted itself */
						this->state = STATE_HOLDING;
					}
					break;

				case STATE_UNHOLDING:
					if(this->cmd.start) {
						i = numArgs;
						this->state = STATE_UNHOLDING;
					}
					break;

				case STATE_SUSPENDING:
					if(this->cmd.suspend) {
						i = numArgs;
						this->internal.pInterrupter = (unsigned long)this; /* module interrupted itself */
						this->state = STATE_SUSPENDING;
					}
					break;

				case STATE_UNSUSPENDING:
					if(this->cmd.start) {
						i = numArgs;
						this->state = STATE_UNSUSPENDING;
					}
					break;

				case STATE_COMPLETING:
					if(this->cmd.complete) {
						i = numArgs;
						this->state = STATE_COMPLETING;
					}
					break;

				case STATE_ABORTING:
					if(this->cmd.abort) {
						i = numArgs;
						this->internal.pInterrupter = (unsigned long)this; /* module interrupted itself */
						this->state = STATE_ABORTING;
					}
					break;

				case STATE_ACTIVATING:
					/* wait for initialization complete */
					if(this->internal.initSubstate == 65000) {
						switch(this->setup.activation) {

							case BRDK_EM_ACTIVATE:
								this->state = STATE_ACTIVATING;
								break;

							case BRDK_EM_ACTIVATE_BY_PARENT:
								if(parent != NULL) {
									switch(parent->state) {
										case STATE_DEACTIVATING: case STATE_DEACTIVATED: brdkStrCpy((unsigned long)this->status.substate,(unsigned long)"waiting for parent's activation"); break;
										default: this->state = STATE_ACTIVATING; break;
									}
								}
							break;

							case BRDK_EM_ACTIVATE_BY_CHILD:
								for(j=0; j <= BRDK_EM_MAX_CHILDREN; j++) {
									child = getEm(this->internal.muList.childrenIdx[j]);
									if(child != NULL) {
										switch(child->state) {
											case STATE_DEACTIVATING: case STATE_DEACTIVATED: brdkStrCpy((unsigned long)this->status.substate,(unsigned long)"waiting for a child's activation"); break;
											default: this->state = STATE_ACTIVATING; break;
										}
									}
								}
								break;

							default:
								brdkStrCpy((unsigned long)this->status.substate,(unsigned long)"waiting for activation");
								break;

						}
					}
					break;

				case STATE_DEACTIVATING:
					switch(this->setup.activation) {

						case BRDK_EM_DEACTIVATE:
							for(j=0; j <= BRDK_EM_MAX_CHILDREN; j++) {		/* check all children */
								child = getEm(this->internal.muList.childrenIdx[j]);
								if(child != NULL) {
									if(child->state != STATE_DEACTIVATED && child->state && STATE_DEACTIVATING) break;
								}
							}
							if(j > BRDK_EM_MAX_CHILDREN) {
								i = numArgs;
								this->state = STATE_DEACTIVATING;
							}
							break;

						case BRDK_EM_ACTIVATE_BY_PARENT:
							if(parent != NULL) {
								switch(parent->state) {
									case STATE_DEACTIVATING: case STATE_DEACTIVATED: this->state = STATE_DEACTIVATING; break;
									default: break;
								}
							}
							break;

						default:
							break;

					}
					break;

				default:
					break;

			}
		}
		va_end(list);
		/* check if an unvalid command has been given */
		this->status.unvalidatedCmd = this->state != this->internal.old.state ? false : this->cmd.abort || this->cmd.clear || this->cmd.stop || this->cmd.reset || this->cmd.start || this->cmd.hold || this->cmd.suspend || this->cmd.complete;
	}
}

/* Add's a child to the parents child list */
unsigned short RegisterChild(brdkEM_typ* this, brdkEM_typ* parent) {
	int i=0, j=0;
	if(parent != NULL) {
		for(i=0; i < BRDK_EM_MAX_CHILDREN; i++) {
			if(parent->internal.muList.childrenIdx[i] == this->internal.muList.idx) break;	/* child already exists in array. index is returned */
			else if(parent->internal.muList.childrenIdx[i] == -1) {							/* finds an empty spot in the array */
				j = SemAcquire(parent->internal.SemCreate_0.ident);							/* checks if the semaphore is free */
				if(j == ERR_OK) {
					parent->internal.muList.childrenIdx[i] = this->internal.muList.idx;		/* puts the index in the array */
					parent->status.childCount++;
					SemRelease(parent->internal.SemCreate_0.ident);							/* releases the semaphore again */
					i = ERR_OK;
				}
				else {
					i = j;	/* 33322: Semaphore with the specified ident does not exist   33323: Semaphore is being used */
					brdkStrCpy((unsigned long)&this->status.substate,(unsigned long)&"semaphore error: ");
					brdkStrAppendUdintToA(j,(unsigned long)&this->status.substate,10,-1);
				}
				break;
			}
		}
		if(i == BRDK_EM_MAX_CHILDREN) {  /* error: child array too small. Solution: make child array bigger */
			brdkStrCpy((unsigned long)&this->status.substate,(unsigned long)&"parent child array full. Increase BRDK_EM_MAX_CHILDREN.");
		}
	}
	return i;
}

/* Unregister a child */
unsigned short UnregisterChild(brdkEM_typ* this, brdkEM_typ* parent) {
	int i=65000,j;
	if(parent != NULL) {
		for(i=0; i < BRDK_EM_MAX_CHILDREN; i++) {
			if(parent->internal.muList.childrenIdx[i] == this->internal.muList.idx) {	/* child found */
				j = SemAcquire(parent->internal.SemCreate_0.ident);	/* checks if the semaphore is free */
				if(j == ERR_OK) {
					parent->internal.muList.childrenIdx[i] = -1;			/* pointer is removed from the array */
					parent->status.childCount--;
					for(j=i; j < BRDK_EM_MAX_CHILDREN; j++) parent->internal.muList.childrenIdx[j] = parent->internal.muList.childrenIdx[j+1];
					SemRelease(parent->internal.SemCreate_0.ident);		/* releases the semaphore again */
					i = ERR_OK;
					this->internal.muList.parentIdx = -1;
				}
				else {
					i = j;	/* 33322: Semaphore with the specified ident does not exist   33323: Semaphore is being used */
					brdkStrCpy((unsigned long)&this->status.substate,(unsigned long)&"semaphore error: ");
					brdkStrAppendUdintToA(j,(unsigned long)&this->status.substate,10,-1);
				}
				break;
			}
		}
		if(i == BRDK_EM_MAX_CHILDREN) {  /* error: child not found in array */
			brdkStrCpy((unsigned long)&this->status.substate,(unsigned long)&"child not found in parent array.");
		}
	}
	return i;
}
```

#### brdkCM.c - Represents a control module.
```c
#include <brdkCM_func.h>

void brdkCM(struct brdkCM* this) {
	int i;
	brdkEM_typ* parent = getEm(this->internal.muList.parentIdx);
	brdk_mu_setup_module_typ module;

	/* initialize control module */
	switch(this->internal.initSubstate) {

		case 0:	/* this substate is only called in void _INIT / PROGRAM _INIT */
			brdkStrCpy((unsigned long)this->status.state,(unsigned long)"initializing - looking for module pointers");
			if(this->setup.name[0] == 0) ST_name(0,(char*)&this->setup.name,(unsigned char)0); 														/* set module name to task name if not set*/
			brdkStrCpy((unsigned long)this->status.name,(unsigned long)this->setup.name);
			if(this->setup.nameIdx > -1) brdkStrAppendUdintToA(this->setup.nameIdx,(unsigned long)&this->status.name, BRDK_STR_CONVERT_DECIMAL,-1);	/* add index to task name */
			this->internal.muList.parentIdx = -1;
			for(i=0; i<= BRDK_MU_MAX_SIBLINGS; i++) this->internal.muList.siblingIdx[i] = -1;
			this->internal.initSubstate = 10;
			break;

		case 10:
			if(!emListReady) brdkStrCpy((unsigned long)this->status.state,(unsigned long)"waiting for mu list to be ready");
			else {
				brdkStrCpy((unsigned long)module.name,(unsigned long)this->setup.name);
				module.index = this->setup.nameIdx;
				this->internal.muList.idx = getMUIndex((unsigned long)this, &module);
				if(this->internal.muList.idx != -1) {
					wakeMU(this->internal.muList.idx,(unsigned long)this);
					if(this->setup.lastActivated) {
						brdkStrMemMove((unsigned long)this->status.last[1],(unsigned long)this->status.last[0], sizeof(this->status.last[0])*BRDK_MU_MAX_LAST_SIZE);
						brdkStrCpy((unsigned long)this->status.last[0],(unsigned long)"module awake");
					}
					this->internal.initSubstate = 65001;
				}
				else {
					if(SemAcquire(SemCreateMUList.ident) != ERR_OK) brdkStrCpy((unsigned long)this->status.state,(unsigned long)"waiting global semaphore to be free");
					else {
						this->internal.muList.idx = addToMUList((unsigned long)this,0);
						SemRelease(SemCreateMUList.ident);
						brdkStrCpy((unsigned long)this->status.state,(unsigned long)"module added em list");
						if(this->internal.muList.idx != -1) this->internal.initSubstate = !this->setup.parent.name[0] ? 40 : 30;	/* check if the module has a parent name assigned */
						else {
							brdkStrCpy((unsigned long)this->status.state,(unsigned long)"em list full. Expand BRDK_EM_MAX_EMS.");
							this->internal.initSubstate = 200;
						}
					}
				}
			}

		case 30:	/* find parent */
			this->internal.muList.parentIdx = getMUIndex((unsigned long)this, &this->setup.parent);
			if(this->internal.muList.parentIdx == -1) brdkStrCpy((unsigned long)this->status.state,(unsigned long)"parent not found");
			else this->internal.initSubstate = 40;
			break;

		case 40:	/* find siblings */
			for(i=0; i<= BRDK_MU_MAX_SIBLINGS; i++) {
				if(this->setup.sibling[i].name[0] != 0) {
					this->internal.muList.siblingIdx[i] = getMUIndex((unsigned long)this, &this->setup.sibling[i]);
					if(this->internal.muList.siblingIdx[i] == -1) {
						brdkStrCpy((unsigned long)this->status.state,(unsigned long)"sibling: ");
						brdkStrCat((unsigned long)this->status.state,(unsigned long)this->setup.sibling[i].name);
						brdkStrCat((unsigned long)this->status.state,(unsigned long)" not found");
						break;
					}
				}
			}
			if(i>=BRDK_MU_MAX_SIBLINGS) {
				this->status.state[0] = 0;	/* reset status text */
				this->internal.initSubstate = 65000;
			}
			break;

		case 65000:	/* module ready */
			/* check if status is not set */
			if(this->status.state[0] == 0) {
				brdkStrUdintToA(this->state,(unsigned long)this->status.state,BRDK_STR_CONVERT_DECIMAL);
				if(this->substate != 0) {
					brdkStrCat((unsigned long)this->status.state,(unsigned long)": ");
					brdkStrAppendUdintToA(this->substate,(unsigned long)this->status.state,BRDK_STR_CONVERT_DECIMAL,-1);
				}
				if(this->description[0] != 0) {
					brdkStrCat((unsigned long)this->status.state,(unsigned long)": ");
					brdkStrCat((unsigned long)this->status.state,(unsigned long)this->description);
				}
			}

			/* state change */
			if(this->state != this->internal.old.state || this->substate != this->internal.old.substate) {
				/* save last state for log */
				if(this->setup.lastActivated) {
					brdkStrMemMove((unsigned long)this->status.last[1],(unsigned long)this->status.last[0], sizeof(this->status.last[0])*BRDK_MU_MAX_LAST_SIZE);
					brdkStrUdintToA(this->internal.old.state,(unsigned long)this->status.last[0],BRDK_STR_CONVERT_DECIMAL);
					brdkStrCat((unsigned long)this->status.last[0],(unsigned long)": ");
					if(this->internal.old.substate || this->substate != 0) {	/* if the substate != 0 then we also want to log the oldsubstate even if it's 0 */
						brdkStrAppendUdintToA(this->internal.old.substate,(unsigned long)this->status.last[0],BRDK_STR_CONVERT_DECIMAL,-1);
						brdkStrCat((unsigned long)this->status.last[0], (unsigned long)": ");
					}
					brdkStrAppendUdintToA(this->status.time, (unsigned long)this->status.last[0],BRDK_STR_CONVERT_DECIMAL,-1);
					brdkStrCat((unsigned long)this->status.last[0], (unsigned long)"ms");
				}
				/* reset */
				if(this->state != this->internal.old.state) this->substate = 0;	/* if the state has been changed the substate will be reset */
				this->status.state[0] = this->description[0] = 0;
				this->internal.old.state = this->state;
				this->internal.old.substate = this->substate;
				this->status.time = 0;
			}
			else this->status.time += this->status.cycleTime/1000;

			/* update parent info */
			if(parent != NULL) {
				this->status.parent.state = parent->state;
				this->status.parent.substate = parent->substate;
				this->status.parent.sleeping = parent->status.sleeping;
				this->status.parent.sc = parent->cmd.sc;
			}

			/* update siblings info */
			updateSiblingInfo(&this->internal.muList.siblingIdx, &this->status.sibling[0]);

			this->status.level = parent != NULL ? parent->status.level+1 : 0;	/* sets the hierarchy level */

			break;

	}

	if(!this->status.cycleTime) this->status.cycleTime = getCycleTime();	/* get the modules cycle time */
	this->status.ready = this->internal.initSubstate == 65000;

}
```

#### brdkCMSleep.c - Put a control module to sleep. It's pointer is added to a sleeping module list where it can be found again by brdkCMWake().
```c
#include <brdkMU_func.h>

signed long brdkCMSleep(unsigned long pCM) {
	brdkCM_typ* this;
	if(pCM != 0) {
		this = (brdkCM_typ*)pCM;
		this->status.sleeping = true;
		if(this->setup.lastActivated) {
			brdkStrMemMove((unsigned long)this->status.last[1],(unsigned long)this->status.last[0], sizeof(this->status.last[0])*BRDK_MU_MAX_LAST_SIZE);
			brdkStrCpy((unsigned long)this->status.last[0],(unsigned long)"module put to sleep");
		}
		return sleepMU(this->internal.muList.idx, pCM);
	}
	return -1;
}
```

- CHANGELOG - brdkMU change log file (not shown)

### Library Logical/Libraries/brdkSIM (ANSIC)
Depends on: AsIO, AsBrStr, sys_lib

#### Types.typ - Exported data types
```iecst
TYPE
	brdkSIM_status_typ : 	STRUCT
		fbStatus : brdkSIM_STATUS_typ;
		error : BOOL;
		errorCode : UINT;
	END_STRUCT;
	brdkSIM_STATUS_typ :
		(
		brdkSIM_NOT_ENABLED := 0,
		brdkSIM_BUSY := 10,
		brdkSIM_RUNNING := 20,
		brdkSIM_ERROR := 200
		);
	brdkSimInput_internal_typ : 	STRUCT
		state : USINT;
		AsIOEnableForcing_0 : AsIOEnableForcing;
		AsIOSetForceValue_0 : AsIOSetForceValue;
		AsIODisableForcing_0 : AsIODisableForcing;
	END_STRUCT;
	brdkSimOutput_internal_typ : 	STRUCT
		state : USINT;
		pvStatus : UINT;
		pvAdr : UDINT;
		pvLen : UDINT;
		pvCheck : UINT;
		pvCmpString : STRING[4];
		boolVar : BOOL;
	END_STRUCT;
END_TYPE
```

#### brdkSimInput.c
```c
#include <bur/plctypes.h>
#include <AsIO.h>
#include <AsBrStr.h>

#ifdef __cplusplus
	extern "C"
	{
#endif
	#include "brdkSIM.h"
#ifdef __cplusplus
	};
#endif

#define false 0
#define true 1

/* TODO: Add your comment here */
void brdkSimInput(struct brdkSimInput* inst)
{
	if (!inst->enable && inst->internal.state > 0 && inst->internal.state < 50) {
		inst->internal.state = 50;
	}

	switch (inst->internal.state) {
		case 0: //wait for enable force
			inst->status.fbStatus = brdkSIM_NOT_ENABLED;
			inst->status.error = false;
			inst->status.errorCode = 0;
			if (inst->enable) {
				inst->internal.state = 10;
			}
			break;

		case 10: //enable force
			inst->status.fbStatus = brdkSIM_BUSY;
			if (!inst->internal.AsIOEnableForcing_0.enable) {
				inst->internal.AsIOEnableForcing_0.enable = true;
				inst->internal.AsIOEnableForcing_0.pDatapoint = (UDINT)&inst->dpName;		// set pointer to the var name (address)
				inst->internal.state = 20;
			}
			break;

		case 20: //wait for AsIOEnableForcing_0 fb to be ready
			if (inst->internal.AsIOEnableForcing_0.status == ERR_OK) {
				inst->internal.AsIOEnableForcing_0.enable = false;					// remember to set enable false so the fb is ready for the next dp
				AsIOEnableForcing(&inst->internal.AsIOEnableForcing_0);
				inst->internal.state = 30;
			}
			else if (inst->internal.AsIOEnableForcing_0.status != ERR_OK && inst->internal.AsIOEnableForcing_0.status != ERR_FUB_BUSY && inst->internal.AsIOEnableForcing_0.status != ERR_FUB_ENABLE_FALSE) {
				inst->status.fbStatus = brdkSIM_ERROR;
				inst->status.error = true;
				inst->status.errorCode = inst->internal.AsIOEnableForcing_0.status;
				inst->internal.state = 200;
			}
			break;

		case 30: //AsIOSetForceValue_0 fb use to control force value
			inst->status.fbStatus = brdkSIM_RUNNING;
			inst->internal.AsIOSetForceValue_0.enable 		= true;
			inst->internal.AsIOSetForceValue_0.pDatapoint	= (UDINT)&inst->dpName;		// set pointer to the dp name (address)
			inst->internal.AsIOSetForceValue_0.value 		= inst->setValue;						// set the force value

			if (inst->internal.AsIOSetForceValue_0.status != ERR_OK && inst->internal.AsIOSetForceValue_0.status != ERR_FUB_BUSY && inst->internal.AsIOSetForceValue_0.status != ERR_FUB_ENABLE_FALSE) {
				inst->status.fbStatus = brdkSIM_ERROR;
				inst->status.error = true;
				inst->status.errorCode = inst->internal.AsIOSetForceValue_0.status;
				inst->internal.state = 200;
			}

			break;

		case 50: //set value to 0 before disable
			inst->status.fbStatus = brdkSIM_BUSY;
			if (inst->internal.AsIOSetForceValue_0.value != 0) {
				inst->internal.AsIOSetForceValue_0.enable 		= true;
				inst->internal.AsIOSetForceValue_0.pDatapoint	= (UDINT)&inst->dpName;		// set pointer to the dp name (address)
				inst->internal.AsIOSetForceValue_0.value 		= 0;									// set the force value

				if (inst->internal.AsIOSetForceValue_0.status != ERR_OK && inst->internal.AsIOSetForceValue_0.status != ERR_FUB_BUSY && inst->internal.AsIOSetForceValue_0.status != ERR_FUB_ENABLE_FALSE) {
					inst->status.fbStatus = brdkSIM_ERROR;
					inst->status.error = true;
					inst->status.errorCode = inst->internal.AsIOSetForceValue_0.status;
					inst->internal.state = 200;
				}
				else {
					inst->internal.state 	= 60;
				}
			}
			else {
				inst->internal.state 	= 60;
			}
			break;

		case 60: //wait for AsIODisableForcing_0 fb to be ready
			inst->internal.AsIOSetForceValue_0.enable 		= false;
			inst->internal.AsIODisableForcing_0.enable 		= true;
			inst->internal.AsIODisableForcing_0.pDatapoint 	= (UDINT)&inst->dpName;		// set pointer to the dp name (address)
			AsIODisableForcing(&inst->internal.AsIODisableForcing_0);

			if (inst->internal.AsIODisableForcing_0.status == ERR_OK) {
				inst->internal.AsIODisableForcing_0.enable 	= false;						// remember to set enable false so the fb is ready for the next dp
				inst->internal.state = 0;
			}
			else if (inst->internal.AsIODisableForcing_0.status != ERR_OK && inst->internal.AsIODisableForcing_0.status != ERR_FUB_BUSY && inst->internal.AsIODisableForcing_0.status != ERR_FUB_ENABLE_FALSE) {
				inst->status.fbStatus = brdkSIM_ERROR;
				inst->status.error = true;
				inst->status.errorCode = inst->internal.AsIODisableForcing_0.status;
				inst->internal.state = 200;
			}
			break;

		case 200: //error
			inst->internal.AsIOEnableForcing_0.enable = false;
			inst->internal.AsIOSetForceValue_0.enable = false;
			inst->internal.AsIODisableForcing_0.enable 	= false;

			if (!inst->enable) {
				inst->status.error = false;
				inst->status.errorCode = 0;
				inst->internal.state 	= 0;
			}
	}

	AsIOEnableForcing(&inst->internal.AsIOEnableForcing_0);
	AsIOSetForceValue(&inst->internal.AsIOSetForceValue_0);
	AsIODisableForcing(&inst->internal.AsIODisableForcing_0);
}
```

#### brdkSimOutput.c
```c
#include <bur/plctypes.h>
#include <sys_lib.h>
#include <AsBrStr.h>

#ifdef __cplusplus
	extern "C"
	{
#endif
	#include "brdkSIM.h"
#ifdef __cplusplus
	};
#endif

#define false 0
#define true 1

/* TODO: Add your comment here */
void brdkSimOutput(struct brdkSimOutput* inst)
{
	if (!inst->enable && inst->internal.state > 0) {
		inst->internal.state = 0;
		inst->internal.pvAdr = 0;
		inst->internal.pvCheck = 0;
		inst->internal.pvLen = 0;
		inst->internal.pvStatus = 0;
		inst->internal.state = 0;
	}

	switch (inst->internal.state) {
		case 0: //wait for enable
			inst->status.fbStatus = brdkSIM_NOT_ENABLED;
			inst->status.error = false;
			inst->status.errorCode = 0;

			if(inst->enable) {
				brsstrcpy((UDINT)inst->internal.pvCmpString, (UDINT) "");
				inst->internal.pvCheck = brsstrcmp((UDINT)inst->pvName, (UDINT)inst->internal.pvCmpString);
				if(inst->internal.pvCheck != 0) {
					inst->internal.state = 10;
				}
				else {
					inst->status.fbStatus = brdkSIM_ERROR;
					inst->status.error = true;
					inst->status.errorCode = 1000;
					inst->internal.state = 200;
				}
			}
			break;

		case 10: //get address of the pv
			inst->status.fbStatus = brdkSIM_BUSY;
			inst->internal.pvStatus = PV_xgetadr(&inst->pvName, &inst->internal.pvAdr, &inst->internal.pvLen);

			if(inst->internal.pvStatus != 0) {
				inst->status.fbStatus = brdkSIM_ERROR;
				inst->status.error = true;
				inst->status.errorCode = inst->internal.pvStatus;
				inst->internal.state = 200;
			}
			else {
				inst->internal.state = 20;
			}
			break;

		case 20: //check value
			inst->status.fbStatus = brdkSIM_RUNNING;
			brsmemcpy((UDINT)&inst->actValue, (UDINT)inst->internal.pvAdr, inst->internal.pvLen);
			break;

		case 200: //error
			break;
	}
}
```

### Library Logical/Libraries/brdkCSV (ANSIC)

#### brdkCSV.fun - Exported functions and function blocks
```iecst
{REDUND_ERROR} FUNCTION brdkSearch : BOOL (*TODO: Add your comment here*) (*$GROUP=User,$CAT=User,$GROUPICON=User.png,$CATICON=User.png*)
	VAR_INPUT
		line : STRING[1000000];
		columnNum : UINT;
		column : UINT;
		row : UINT;
		result : STRING[255];
	END_VAR
END_FUNCTION
```

#### brdkSearch.c
```c
#include <bur/plctypes.h>
#include <string.h>

#ifdef __cplusplus
	extern "C"
	{
#endif
	#include "brdkCSV.h"
#ifdef __cplusplus
	};
#endif
/* TODO: Add your comment here */
plcbit brdkSearch(plcstring* line, unsigned short columnNum, unsigned short column, unsigned short row, plcstring* result)
{

	signed long idx = 0;
	unsigned long size = (row * columnNum) + column;
	plcstring* tok;
//	char internal[100];

//	strcpy(internal, line);

	tok = strtok(line, ";");

	if(size == 0){
		strcpy(result, tok);
		return 1;
	}

	/* walk through other tokens */
	while( tok != NULL ) {
		tok = strtok(NULL, ";");
		idx++;
		if(idx >= size){
			strcpy(result, tok);
			return 1;
		}
	}

	return NULL;
}
```

### Library Logical/Libraries/brdkPV (ANSIC, version 1.00.0) - PV handling library.
Depends on: brdkSTR, sys_lib

#### brdkPV.var
```iecst
VAR CONSTANT
	BRDK_PV_MAX_NAME_LENGTH : UINT := 80; (*Max length of string containing the variable names.*)
	BRDK_PV_MAX_PV_NAMES : UINT := 9; (*9 means 10 elements*)
END_VAR
```

#### brdkPV.fun
```iecst
FUNCTION_BLOCK brdkPVLocalVariable (*Creates the PV names for the variables which can be used for e.g. mappRecipe or mappData.*) (*$GROUP=User,$CAT=User,$GROUPICON=User.png,$CATICON=User.png*)
	VAR_INPUT
		pPV : ARRAY[0..BRDK_PV_MAX_PV_NAMES] OF UDINT := [10(0)]; (*String pointer for each variable.*)
		lPV : ARRAY[0..BRDK_PV_MAX_PV_NAMES] OF STRING[BRDK_PV_MAX_NAME_LENGTH] := [10('')]; (*String list of local variables.*)
	END_VAR
	VAR_OUTPUT
		status : UINT := 0; (*Status of the function block.*)
	END_VAR
END_FUNCTION_BLOCK
```

#### brdkPVLocalName.c
```c
#include <brdkPV_func.h>

void brdkPVLocalVariable(struct brdkPVLocalVariable* this)
{
	char taskName[20];
	ST_name(0,(char*)&taskName,0);
	brdkStrCat((unsigned long)&taskName,(unsigned long)&":");
	unsigned short i = 0;
	unsigned long adr, length;
	this->status = 0;

	/* create the strings */
	for(;i < BRDK_PV_MAX_PV_NAMES; i++) {
		if(this->pPV[i] != 0) {
			brdkStrCpy((unsigned long)&this->lPV[i],(unsigned long)&taskName);
			brdkStrCat((unsigned long)&this->lPV[i],this->pPV[i]);
			this->status = PV_xgetadr((char*)&this->lPV[i],&adr,&length);
			/* check that the variable exists */
			if(this->status != 0) brdkStrCpy((unsigned long)&this->lPV[i],(unsigned long)&"PV not found. Check spelling");
		}
	}
}
```

#### brdkPV_func.h
```c
#ifndef BRDK_PV_FUNCS
#define BRDK_PV_FUNCS 1

#include <brdkPV.h>
#include <bur/plctypes.h>

#ifdef __cplusplus
	extern "C"
	{
#endif

#ifdef __cplusplus
	};
#endif

#endif
```

#### brdkPV_func.c
```c
#include <brdkPV_func.h>
```

- CHANGELOG - brdkPV change log (not shown)

### Library Logical/Libraries/legoCM20 (IEC)

#### legocm20.typ - Exported data types
```iecst
TYPE
	legocm20_flap_internal_typ : 	STRUCT  (*Flap internal variables.*)
		state : DINT; (*State of the function block.*)
		timeElapsed : UDINT; (*Time elapsed.*)
		startMeasTimeOpenClose : BOOL;
		avgOpenTime : MTFilterMovingAverage;
		avgCloseTime : MTFilterMovingAverage;
		openTimeMaxCnt : USINT;
		closeTimeMaxCnt : USINT;
		openCloseTime : UDINT;
	END_STRUCT;
	legocm20_flap_position_typ :
		( (*Flap positions.*)
		FLAP_OPENING_BEFORE_CHANGEOVER := 1, (*Before changeover.*)
		FLAP_OPENING_AT_CHANGEOVER := 3, (*At changeover.*)
		FLAP_OPEN := 4, (*Open.*)
		FLAP_CLOSEING_BEFORE_CHANGEOVER := 5, (*Before changeover.*)
		FLAP_CLOSEING_AT_CHANGEOVER := 7, (*At changeover.*)
		FLAP_CLOSED := 8 (*Closed.*)
		);
	LEGO_SPEED_ENUM :
		(
		lego_speed_stop := 0,
		lego_speed_wait := 1,
		lego_speed_counting := 2
		);
END_TYPE
```

#### legoCM20.fun - Exported functions and function blocks
```iecst
FUNCTION_BLOCK legoCM20Flap (*Function block for controlling a flap*) (*$GROUP=User,$CAT=User,$GROUPICON=User.png,$CATICON=User.png*)
	VAR_INPUT
		enable : BOOL;
		close : BOOL := FALSE; (*Close the flap.*)
		open : BOOL := FALSE; (*Open the flap.*)
		resetError : BOOL;
		di_changeover : BOOL := FALSE; (*Changeover sensor.*)
		flapTime : UDINT := 0; (*Flap movement time.*)
		cycleTime : UDINT := 0; (*Current cycletime.*)
		avgSamples : USINT := 10;
		WUstepperConnected : BOOL;
		simulation : BOOL;
		positionFromWUstepper : legocm20_flap_position_typ; (*8=FLAP_CLOSED, 4=FLAP_OPEN*)
	END_VAR
	VAR_OUTPUT
		position : legocm20_flap_position_typ := FLAP_CLOSED; (*Actual position of the flap.*)
		do_open : BOOL := FALSE; (*Move flap command.*)
		error : BOOL := FALSE; (*Error. Is removed by a new open or close signal.*)
		closingTime : UDINT;
		openTime : UDINT;
		closingTimeAfterChangeover : UDINT;
		openTimeAfterChangeover : UDINT;
		openCloseTime : UDINT;
	END_VAR
	VAR
		internal : legocm20_flap_internal_typ; (*Internal variables.*)
		TON_0 : TON;
		simulatedTimeToOpenCloseFlap : TIME := T#150ms;
	END_VAR
END_FUNCTION_BLOCK
```

#### legoCM20Flap.st
```iecst
FUNCTION_BLOCK legoCM20Flap

	// open								close
	//  ____________________________________
	// |____________________________________|
	//              /changeover\
	internal.avgOpenTime.Enable := TRUE;
	internal.avgCloseTime.Enable := TRUE;

	IF avgSamples <> internal.avgOpenTime.WindowLength THEN
		internal.avgOpenTime.Update := TRUE;
		internal.avgOpenTime.WindowLength  := avgSamples;

	END_IF

	IF avgSamples <> internal.avgCloseTime.WindowLength THEN
		internal.avgCloseTime.Update := TRUE;
		internal.avgCloseTime.WindowLength  := avgSamples;

	END_IF

	IF internal.avgOpenTime.UpdateDone THEN
		internal.avgOpenTime.Update := FALSE;
	END_IF

	IF internal.avgCloseTime.UpdateDone THEN
		internal.avgCloseTime.Update := FALSE;
	END_IF

	CASE internal.state OF

		0:	// waiting for a start command
			IF NOT enable THEN
				do_open := FALSE;
				internal.state := 100;
			ELSIF WUstepperConnected THEN
				internal.state := 200;
			ELSIF open THEN
				open 					:= FALSE;
				IF simulation THEN
					TON_0(IN:=FALSE);
					open := TRUE;
					internal.state := 110;
				ELSIF position <> FLAP_OPEN THEN
					error					:= FALSE;
					do_open				:= TRUE;					// start opening the flap
					internal.timeElapsed 	:= 0;						// reset elapsed time
					internal.openCloseTime	:= 0;
					internal.startMeasTimeOpenClose := TRUE;
					position				:= FLAP_OPENING_BEFORE_CHANGEOVER;
					internal.state 			:= 10;
				END_IF
			ELSIF close THEN
				close 					:= FALSE;
				IF simulation THEN
					TON_0(IN:=FALSE);
					internal.state := 110;
				ELSIF position <> FLAP_CLOSED THEN
					error					:= FALSE;
					do_open				:= FALSE;					// start closeing the flap
					internal.timeElapsed 	:= 0;						// reset elapsed time
					position				:= FLAP_CLOSEING_BEFORE_CHANGEOVER;
					internal.state 			:= 10;
				END_IF
			ELSIF error THEN
				do_open					:= FALSE;
				IF resetError THEN
					internal.timeElapsed 	:= 0;
					internal.state 			:= 40;
				END_IF
			END_IF

		10:	// waiting for changeover sensor
			internal.timeElapsed := internal.timeElapsed + cycleTime;
			IF internal.timeElapsed >= flapTime THEN
				internal.state 	:= 0;
				error			:= TRUE;
			ELSIF NOT di_changeover THEN	 // high signal (active low)
				IF do_open THEN
					IF internal.timeElapsed > REAL_TO_UDINT(internal.avgOpenTime.Out) THEN
						internal.openTimeMaxCnt := internal.openTimeMaxCnt+1;
					ELSE
						internal.openTimeMaxCnt := 0;
					END_IF

					internal.avgOpenTime(In := UDINT_TO_REAL(internal.timeElapsed));
					openTime := internal.timeElapsed;
					position		:= FLAP_OPENING_AT_CHANGEOVER;
				ELSE
					IF internal.timeElapsed > REAL_TO_UDINT(internal.avgCloseTime.Out) THEN
						internal.closeTimeMaxCnt := internal.closeTimeMaxCnt+1;
					ELSE
						internal.closeTimeMaxCnt := 0;
					END_IF

					internal.avgCloseTime(In := UDINT_TO_REAL(internal.timeElapsed));
					internal.startMeasTimeOpenClose := FALSE;
					openCloseTime := internal.openCloseTime;
					closingTime := internal.timeElapsed;
					position		:= FLAP_CLOSEING_AT_CHANGEOVER;
				END_IF

				IF internal.openTimeMaxCnt > 25THEN
					internal.openTimeMaxCnt := 0;
					internal.state 	:= 0;
					error			:= TRUE;
				END_IF

				IF internal.closeTimeMaxCnt > 25THEN
					internal.closeTimeMaxCnt := 0;
					internal.state 	:= 0;
					error			:= TRUE;
				END_IF

				internal.state 	:= 20;
			END_IF

		20:	// waiting for no changeover sensor
			internal.timeElapsed := internal.timeElapsed + cycleTime;
			IF internal.timeElapsed >= flapTime THEN
				internal.state 	:= 0;
				error			:= TRUE;
			ELSIF di_changeover THEN
				position		:= SEL(NOT do_open,FLAP_OPEN,FLAP_CLOSED);
				IF do_open THEN
					openTimeAfterChangeover := (internal.timeElapsed-cycleTime)/1000; // subtract 1 scan because we PVmap from sampling task (takes 1 extra scan).
				ELSE //closing
					closingTimeAfterChangeover := (internal.timeElapsed-cycleTime)/1000;
				END_IF
				internal.state 	:= 0;
			END_IF

		40:
			internal.timeElapsed := internal.timeElapsed + cycleTime;
			IF internal.timeElapsed >= 2*flapTime THEN
				resetError 	:= FALSE;
				position	:= FLAP_CLOSED;
				do_open 	:= FALSE;
				error		:= FALSE;
				internal.state 	:= SEL(WUstepperConnected,0,200);
			END_IF

		100:
			IF enable THEN
				internal.state := SEL(WUstepperConnected,0,200);
			ELSE
				IF open THEN
					open := FALSE;
					position := FLAP_OPEN;
				ELSIF close THEN
					close := FALSE;
					position := FLAP_CLOSED;
				END_IF
			END_IF

		110:
			TON_0.IN := TRUE;
			TON_0.PT := simulatedTimeToOpenCloseFlap;
			TON_0();

			IF TON_0.Q THEN
				TON_0(IN:=FALSE);
				position := SEL(open,FLAP_CLOSED,FLAP_OPEN);
				open := FALSE;
				internal.state := 0;
			END_IF

		(**** STEPPER WU20 ****)

		200:
			IF NOT enable THEN
				do_open := FALSE;
				internal.state := 100;
			ELSIF open THEN
				open 					:= FALSE;
				IF positionFromWUstepper <> FLAP_OPEN THEN
					error					:= FALSE;
					do_open				:= TRUE;						// start opening the flap
					internal.timeElapsed 	:= 0;						// reset elapsed time
					position := FLAP_OPENING_AT_CHANGEOVER;
					internal.state 			:= 210;
				ELSE
					position := FLAP_OPEN;
				END_IF
			ELSIF close THEN
				close 					:= FALSE;
				IF positionFromWUstepper <> FLAP_CLOSED THEN
					error					:= FALSE;
					do_open				:= FALSE;					// start closeing the flap
					internal.timeElapsed 	:= 0;						// reset elapsed time
					position := FLAP_CLOSEING_AT_CHANGEOVER;
					internal.state 			:= 210;
				ELSE
					position := FLAP_CLOSED;
				END_IF
			ELSIF error THEN
				do_open					:= FALSE;
				IF resetError THEN
					internal.timeElapsed 	:= 0;
					internal.state 			:= 40;
				END_IF
			END_IF

		210:
			internal.timeElapsed := internal.timeElapsed + cycleTime;

			IF internal.timeElapsed >= flapTime THEN
				internal.state 	:= 200;
				error			:= TRUE;
			ELSIF (do_open AND positionFromWUstepper=FLAP_OPEN) OR (NOT do_open AND positionFromWUstepper=FLAP_CLOSED) THEN
				position := positionFromWUstepper;
				// Only for timings to show on HMI:
				IF do_open THEN
					openTimeAfterChangeover := (internal.timeElapsed-cycleTime)/1000; // subtract 1 scan because we PVmap from sampling task (takes 1 extra scan).
				ELSE //closing
					closingTimeAfterChangeover := (internal.timeElapsed-cycleTime)/1000;
				END_IF
				internal.state 	:= 200;
			END_IF

	END_CASE

	IF internal.startMeasTimeOpenClose THEN
		internal.openCloseTime := internal.openCloseTime + cycleTime;
	END_IF

END_FUNCTION_BLOCK
```

### Library Logical/Libraries/legoSTR (ANSIC) - Lego Str library

#### Types.typ - Exported data types
```iecst
TYPE
	legoSTRItem_internal : 	STRUCT
		length : UINT; (*Length of the string*)
	END_STRUCT;
END_TYPE
```

#### Constants.var - Exported constants
```iecst
VAR CONSTANT
	MAX_ITEM_SIZE : UINT := 200; (*Max. size of item string*)
END_VAR
```

#### legoSTR.fun - Exported functions and function blocks
```iecst
{REDUND_ERROR} FUNCTION_BLOCK legoSTRItemString (*Outputs an item string*) (*$GROUP=User,$CAT=User,$GROUPICON=User.png,$CATICON=User.png*)
	VAR_INPUT
		trigger : BOOL; (*Trigger *)
		value : USINT; (*Value. [0-9], 20 = BACKSPACE 30 = CLEAR*)
	END_VAR
	VAR_OUTPUT
		item : STRING[MAX_ITEM_SIZE]; (*Item number*)
		internal : legoSTRItem_internal; (*Internal variables*)
	END_VAR
END_FUNCTION_BLOCK
```

#### legoSTRItemString.c
```c
#include <bur/plctypes.h>
#ifdef __cplusplus
	extern "C"
	{
#endif
	#include "legoSTR.h"
#ifdef __cplusplus
	};
#endif
/* Outputs an item string */
void legoSTRItemString(struct legoSTRItemString* inst) {
	legoSTRItem_internal* this = &inst->internal;

	if(inst->trigger) {
		inst->trigger = 0;

		switch(inst->value) {

			case 0 ... 9:
				if(this->length < MAX_ITEM_SIZE) {
					inst->item[this->length] = 0x30 + inst->value;
					this->length++;
				}
				break;

			case 20:	/* BACKSPACE */
				if(this->length > 0) {
					inst->item[this->length-1] = 0;
					this->length--;
				}
				break;

			case 30:	/* CLEAR */
				while(this->length > 0) {
					inst->item[this->length-1] = 0;
					this->length--;
				}
				break;

			default:
				break;

		}

	}
}
```

### Library Logical/Libraries/brdkOPCUA (ANSIC, version 0.00.1) - OPC-UA wrapper library.
Depends on: AsOpcUac, AsOpcUas, brdkSTR

#### brdkOPCUA.typ - Exported data types
```iecst
TYPE
	brdk_opcua_method_op_int_typ : 	STRUCT  (*Internal variables for brdkOPCUAMethodOperate function block.*)
		UaSrv_MethodOperate_0 : UaSrv_MethodOperate; (*UaSrv_MethodOperate.*)
		state : DINT; (*State.*)
	END_STRUCT;
	brdk_opcua_method_op_state_typ :
		( (*Method state type.*)
		BRDK_OPCUA_METHOD_NOT_ENABLED := 0,
		BRDK_OPCUA_METHOD_ERROR := 1,
		BRDK_OPCUA_METHOD_WAIT_FOR_CALL := 2,
		BRDK_OPCUA_METHOD_IS_CALLED := 3,
		BRDK_OPCUA_METHOD_NO_NAME_SET := 4,
		BRDK_OPCUA_METHOD_FINISHING := 5
		);
	brdk_opcua_event_internal_typ : 	STRUCT  (*Internal variables for brdkOPCUAMethodOperate function block.*)
		UaSrv_GetNamespaceIndex_0 : UaSrv_GetNamespaceIndex; (*UaSrv_GetNamespaceIndex.*)
		UaSrv_FireEvent_0 : UaSrv_FireEvent; (*UaSrv_FireEvent.*)
		state : DINT; (*State.*)
		opcNSidx : UINT; (*Namespace index of OPC UA.*)
		pvNSidx : UINT; (*Namespace index of the PV.*)
		plcNSidx : UINT; (*Namespace index of the PLC.*)
		eventFields : ARRAY[0..4]OF UaSrv_FireEventFieldType; (*Event fields.*)
		eventFieldCnt : USINT; (*Event field count.*)
	END_STRUCT;
END_TYPE
```

#### brdkOPCUA.var - Exported constants
```iecst
VAR CONSTANT
	BRDK_OPCUA_MAX_EVENT_NS : USINT := 3; (*3 means 4*)
	BRDK_OPCUA_EVENT_NS_OPCUA : UINT := 4; (*Namespace index of http://opcfoundation.org/UA/*)
	BRDK_OPCUA_EVENT_NS_PV : UINT := 5; (*Namespace index of http://br-automation.com/OpcUa/PLC/PV/*)
	BRDK_OPCUA_EVENT_NS_PLC : UINT := 6; (*Namespace index of http://br-automation.com/OpcUa/PLC/*)
END_VAR
```

#### brdkOPCUA.fun - Exported functions and function blocks
```iecst
FUNCTION_BLOCK brdkOPCUAMethodOperate (*Wrapper function block for operating OPC UA method calls.*) (*$GROUP=User,$CAT=User,$GROUPICON=User.png,$CATICON=User.png*)
	VAR_INPUT
		enable : BOOL; (*Enables the function block.*)
		name : STRING[255]; (*Name of the method to be operated.*)
		finish : BOOL; (*Command to finish the OPC UA method operation. THis is set after receiving an isCalled status.*)
	END_VAR
	VAR_OUTPUT
		state : brdk_opcua_method_op_state_typ; (*State of the method.*)
		errorID : DWORD; (*Error code in the event of error. See OPC UA StatusCode.*)
	END_VAR
	VAR
		internal : brdk_opcua_method_op_int_typ; (*Internal variables.*)
	END_VAR
END_FUNCTION_BLOCK

FUNCTION_BLOCK brdkOPCUAFireEvent (*Wrapper function block for fireing OPC UA events.*) (*$GROUP=User,$CAT=User,$GROUPICON=User.png,$CATICON=User.png*)
	VAR_INPUT
		enable : BOOL; (*Enables the function block.*)
		instanceName : STRING[80]; (*Functioan block instance name.*)
		namespaceUri : ARRAY[0..BRDK_OPCUA_MAX_EVENT_NS] OF STRING[MAX_LENGTH_NAMESPACEURI]; (*Additional namepsace URI's. http://opcfoundation.org/UA/ and http://br-automation.com/OpcUa/PLC/ are defaults.*)
		sourceNode : UANodeID; (*SourceNode identifies the Node that the Event originated from. If the Event is not specific to a Node the NodeId is set to null or not assigned at all. Some subtypes of this BaseEventType may define additional rules for SourceNode.*)
		sourceName : STRING[255]; (*SourceName provides a description of the source of the Event. If the field is not assigned the default value will be set to the DisplayName of the source node.*)
		message : UALocalizedText; (*Event message.*)
		severity : UINT; (*Event severity. Must be between 1 and 1000.*)
		fireEvent : BOOL; (*Fire an event.*)
	END_VAR
	VAR_OUTPUT
		ready : BOOL; (*Ready to fire an event.*)
		errorID : DWORD; (*Error code in the event of error. See OPC UA StatusCode.*)
	END_VAR
	VAR
		internal : brdk_opcua_event_internal_typ; (*Internal variables.*)
	END_VAR
END_FUNCTION_BLOCK
```

#### brdkOPCUAFireEvent.c - Fires an event.
```c
#include <brdkOPCUA_func.h>

void brdkOPCUAFireEvent(struct brdkOPCUAFireEvent* inst) {
	brdk_opcua_event_internal_typ* this = (brdk_opcua_event_internal_typ*)&inst->internal;
	if(inst->enable) {
		switch(this->state) {

			case 0: /* setup get name space index */
				this->UaSrv_GetNamespaceIndex_0.Execute 		= true;
				brdkStrCpy((unsigned long)&(this->UaSrv_GetNamespaceIndex_0.NamespaceUri),(unsigned long)&("http://opcfoundation.org/UA/"));
				this->state = 10;
				break;

			case 10: /* waiting for namespace index */
				UaSrv_GetNamespaceIndex(&this->UaSrv_GetNamespaceIndex_0);
				if(!this->UaSrv_GetNamespaceIndex_0.Error) {
					if(this->UaSrv_GetNamespaceIndex_0.Done) {
						this->opcNSidx = this->UaSrv_GetNamespaceIndex_0.NamespaceIndex;
						this->UaSrv_GetNamespaceIndex_0.Execute = false;
						UaSrv_GetNamespaceIndex(&this->UaSrv_GetNamespaceIndex_0);
						this->UaSrv_GetNamespaceIndex_0.Execute = true;
						brdkStrCpy((unsigned long)&(this->UaSrv_GetNamespaceIndex_0.NamespaceUri),(unsigned long)&("http://br-automation.com/OpcUa/PLC/"));
						this->state = 20;
					}
				}
				else {
					inst->errorID = this->UaSrv_GetNamespaceIndex_0.ErrorID;
				}
				break;

			case 20: /* waiting for namespace index */
				UaSrv_GetNamespaceIndex(&this->UaSrv_GetNamespaceIndex_0);
				if(!this->UaSrv_GetNamespaceIndex_0.Error) {
					if(this->UaSrv_GetNamespaceIndex_0.Done) {
						this->plcNSidx = this->UaSrv_GetNamespaceIndex_0.NamespaceIndex;
						this->UaSrv_GetNamespaceIndex_0.Execute = false;
						UaSrv_GetNamespaceIndex(&this->UaSrv_GetNamespaceIndex_0);
						this->UaSrv_GetNamespaceIndex_0.Execute = true;
						brdkStrCpy((unsigned long)&(this->UaSrv_GetNamespaceIndex_0.NamespaceUri),(unsigned long)&("http://br-automation.com/OpcUa/PLC/PV/"));
						this->state = 30;
					}
				}
				else {
					inst->errorID = this->UaSrv_GetNamespaceIndex_0.ErrorID;
				}
				break;

			case 30: /* waiting for namespace index */
				UaSrv_GetNamespaceIndex(&this->UaSrv_GetNamespaceIndex_0);
				if(!this->UaSrv_GetNamespaceIndex_0.Error) {
					if(this->UaSrv_GetNamespaceIndex_0.Done) {
						this->pvNSidx = this->UaSrv_GetNamespaceIndex_0.NamespaceIndex;
						this->UaSrv_GetNamespaceIndex_0.Execute = false;
						UaSrv_GetNamespaceIndex(&this->UaSrv_GetNamespaceIndex_0);
						this->UaSrv_FireEvent_0.EventFieldCount = 0;

						/* check if a source node should be added */
						if(!brdkStrIsEmpty((unsigned long)&inst->sourceNode.Identifier)) {
							switch(inst->sourceNode.NamespaceIndex) {
								case BRDK_OPCUA_EVENT_NS_OPCUA: inst->sourceNode.NamespaceIndex = this->opcNSidx; break;
								case BRDK_OPCUA_EVENT_NS_PV: inst->sourceNode.NamespaceIndex = this->pvNSidx; break;
								case BRDK_OPCUA_EVENT_NS_PLC: inst->sourceNode.NamespaceIndex = this->plcNSidx; break;

								default:
									//inst->sourceNode.NamespaceIndex = this->;
									break;

							}

							brdkStrCpy((unsigned long)&this->eventFields[this->UaSrv_FireEvent_0.EventFieldCount].BrowsePath,(unsigned long)&"/SourceNode");
							brdkStrCpy((unsigned long)&this->eventFields[this->UaSrv_FireEvent_0.EventFieldCount].Variable,(unsigned long)&inst->instanceName);
							brdkStrCat((unsigned long)&this->eventFields[this->UaSrv_FireEvent_0.EventFieldCount].Variable,(unsigned long)&".sourceNode");
							this->UaSrv_FireEvent_0.EventFieldCount++;
						}

						/* check if a source name should be added */
						if(!brdkStrIsEmpty((unsigned long)&inst->sourceName)) {
							brdkStrCpy((unsigned long)&this->eventFields[this->UaSrv_FireEvent_0.EventFieldCount].BrowsePath,(unsigned long)&"/SourceName");
							brdkStrCpy((unsigned long)&this->eventFields[this->UaSrv_FireEvent_0.EventFieldCount].Variable,(unsigned long)&inst->instanceName);
							brdkStrCat((unsigned long)&this->eventFields[this->UaSrv_FireEvent_0.EventFieldCount].Variable,(unsigned long)&".sourceName");
							this->UaSrv_FireEvent_0.EventFieldCount++;
						}

						/* check if a message should be added */
						if(!brdkStrIsEmpty((unsigned long)&inst->message.Text)) {
							brdkStrCpy((unsigned long)&this->eventFields[this->UaSrv_FireEvent_0.EventFieldCount].BrowsePath,(unsigned long)&"/Message");
							brdkStrCpy((unsigned long)&this->eventFields[this->UaSrv_FireEvent_0.EventFieldCount].Variable,(unsigned long)&inst->instanceName);
							brdkStrCat((unsigned long)&this->eventFields[this->UaSrv_FireEvent_0.EventFieldCount].Variable,(unsigned long)&".message");
							this->UaSrv_FireEvent_0.EventFieldCount++;
						}

						/* check is severity should be added */
						if(inst->severity > 0 && inst->severity < 1001) {
							brdkStrCpy((unsigned long)&this->eventFields[this->UaSrv_FireEvent_0.EventFieldCount].BrowsePath,(unsigned long)&"/Severity");
							brdkStrCpy((unsigned long)&this->eventFields[this->UaSrv_FireEvent_0.EventFieldCount].Variable,(unsigned long)&inst->instanceName);
							brdkStrCat((unsigned long)&this->eventFields[this->UaSrv_FireEvent_0.EventFieldCount].Variable,(unsigned long)&".severity");
							this->UaSrv_FireEvent_0.EventFieldCount++;
						}

						this->UaSrv_FireEvent_0.EventType.NamespaceIndex = this->opcNSidx;
						this->UaSrv_FireEvent_0.EventType.IdentifierType = UAIdentifierType_Numeric;
						brdkStrCpy((unsigned long)&this->UaSrv_FireEvent_0.EventType.Identifier,(unsigned long)&"2041");
						this->UaSrv_FireEvent_0.EventFields = this->eventFields;
						inst->ready = true;
						this->state = 100;
					}
				}
				else {
					inst->errorID = this->UaSrv_GetNamespaceIndex_0.ErrorID;
				}
				break;

			case 100:
				this->UaSrv_FireEvent_0.Execute = inst->fireEvent;
				UaSrv_FireEvent(&this->UaSrv_FireEvent_0);
				if(!this->UaSrv_FireEvent_0.Error) {
					if(this->UaSrv_FireEvent_0.Done) {
						inst->fireEvent = false;
						this->UaSrv_FireEvent_0.Execute = false;
						UaSrv_FireEvent(&this->UaSrv_FireEvent_0);
					}
				}
				break;

		}
	}
	else {
		inst->ready = false;
		this->UaSrv_FireEvent_0.Execute = false;
		UaSrv_FireEvent(&this->UaSrv_FireEvent_0);
	}
}
```

#### brdkOPCUAMethodOperate.c - Operates a method.
```c
#include <brdkOPCUA_func.h>

void brdkOPCUAMethodOperate(struct brdkOPCUAMethodOperate* inst) {
	brdk_opcua_method_op_int_typ* this = (brdk_opcua_method_op_int_typ*)&inst->internal;
	if(inst->enable) {
		switch(this->state) {

			case 0:	/* checking that the name is different from empty */
				if(!brdkStrIsEmpty((unsigned long)inst->name)) {
					brdkStrCpy((unsigned long)&this->UaSrv_MethodOperate_0.MethodName,(unsigned long)inst->name);
					inst->state = BRDK_OPCUA_METHOD_WAIT_FOR_CALL;
					this->state = 10;
				}
				else inst->state = BRDK_OPCUA_METHOD_NO_NAME_SET;
				break;

			case 10: /* waiting for UaSrv_MethodOperate_0 to be done */
				this->UaSrv_MethodOperate_0.Execute = false;
				UaSrv_MethodOperate(&this->UaSrv_MethodOperate_0);
				if(!this->UaSrv_MethodOperate_0.Done) {
					this->state = 11;
				}
				break;

			case 11:
				this->UaSrv_MethodOperate_0.Execute = !this->UaSrv_MethodOperate_0.Busy;
				this->UaSrv_MethodOperate_0.Action = UaMoa_CheckIsCalled;
				UaSrv_MethodOperate(&this->UaSrv_MethodOperate_0);
				if(!this->UaSrv_MethodOperate_0.Error) {
					if(this->UaSrv_MethodOperate_0.Done) {
						inst->state = BRDK_OPCUA_METHOD_WAIT_FOR_CALL; // If FB done - we don't have an error anymore.
						if(this->UaSrv_MethodOperate_0.IsCalled) {
							inst->state = BRDK_OPCUA_METHOD_IS_CALLED;
							this->state = 20;
						}
						else {
							this->state = 10;
						}
					}
				}
				else {
					inst->state = BRDK_OPCUA_METHOD_ERROR;
					inst->errorID = this->UaSrv_MethodOperate_0.ErrorID;
				}
				break;

			case 20:	/* waiting for finish command */
				if(inst->finish) {
					inst->finish = false;
					this->UaSrv_MethodOperate_0.Execute = true;
					this->UaSrv_MethodOperate_0.Action = UaMoa_Finished;
					UaSrv_MethodOperate(&this->UaSrv_MethodOperate_0);
					if(!this->UaSrv_MethodOperate_0.Error) {
						inst->state = BRDK_OPCUA_METHOD_FINISHING;
						if(this->UaSrv_MethodOperate_0.Done) {
							inst->state = BRDK_OPCUA_METHOD_WAIT_FOR_CALL;
							this->UaSrv_MethodOperate_0.Execute = false;
							UaSrv_MethodOperate(&this->UaSrv_MethodOperate_0);
							this->state = 10;
						}
						else {
							this->state = 30;
						}
					}
					else {
						inst->state = BRDK_OPCUA_METHOD_ERROR;
						inst->errorID = this->UaSrv_MethodOperate_0.ErrorID;
					}
				}
				break;

			case 30: /* waiting for UaSrv_MethodOperate_0 to be done */
				UaSrv_MethodOperate(&this->UaSrv_MethodOperate_0);
				if(!this->UaSrv_MethodOperate_0.Error) {
					if(this->UaSrv_MethodOperate_0.Done) {
						inst->state = BRDK_OPCUA_METHOD_WAIT_FOR_CALL;
						this->UaSrv_MethodOperate_0.Execute = false;
						UaSrv_MethodOperate(&this->UaSrv_MethodOperate_0);
						this->state = 10;
					}
				}
				else {
					inst->state = BRDK_OPCUA_METHOD_ERROR;
					inst->errorID = this->UaSrv_MethodOperate_0.ErrorID;
				}
				break;

		}
	}
	else {
		this->UaSrv_MethodOperate_0.Execute = false;
		UaSrv_MethodOperate(&this->UaSrv_MethodOperate_0);
		inst->state = BRDK_OPCUA_METHOD_NOT_ENABLED;
	}
}
```

#### brdkOPCUA_func.h - Header for internal functions for brdkOPCUA.
```c
#ifndef BRDK_OPCUA_FUNCS
#define BRDK_OPCUA_FUNCS 1

#include <brdkOPCUA.h>
#include <bur/plctypes.h>

#ifdef __cplusplus
	extern "C"
	{
#endif

#ifdef __cplusplus
	};
#endif

#define false 0
#define true 1

#endif /* !BRDK_OPCUA_FUNCS */
```

#### brdkOPCUA_func.c - Internal functions for brdkOPCUA.
```c
#include <brdkOPCUA_func.h>
```

- CHANGELOG (not shown)

### Library Logical/Libraries/brdkUpdate (ANSIC, version 1.00.0) - This library handles updates.
Depends on: ArProject, brdkSTR, FileIO, brdkFile, AsIODiag, sys_lib

#### brdkUpdate.typ - Exported data types
```iecst
TYPE
	brdk_update_manager_internal_typ : 	STRUCT  (*Manager internal variables.*)
		state : DINT := 0; (*Internal state.*)
		ArProjectGetInfo_0 : ArProjectGetInfo; (*ArProjectGetInfo.*)
		ArProjectInstallPackage_0 : ArProjectInstallPackage; (*ArProjectInstallPackage.*)
		versionCmp : DINT := 0; (*Version compare.*)
		brdkUpdateCheck_0 : brdkUpdateCheck; (*brdkUpdateCheck.*)
		brdkUpdateDelete_0 : brdkUpdateDelete; (*brdkUpdateDelete.*)
	END_STRUCT;
	brdk_update_manager_run_info_typ : 	STRUCT  (*Information.*)
		id : STRING[255] := ''; (*Unique machine ID.*)
		version : STRING[32] := ''; (*Machine version.*)
	END_STRUCT;
	brdk_update_manager_upd_info_typ : 	STRUCT  (*Information.*)
		status : brdk_update_manager_upd_stat_typ := BRDK_UPDATE_NOT_FOUND; (*Indicates if an update is found on the flash.*)
		id : STRING[255] := ''; (*Unique machine ID.*)
		version : STRING[32] := ''; (*Machine version.*)
		artransferFileSize : UDINT := 0; (*File size of "artransfer.br" in bytes.*)
	END_STRUCT;
	brdk_update_manager_upd_stat_typ :
		( (*Status of the update package.*)
		BRDK_UPDATE_NOT_FOUND := 0, (*Update package not found.*)
		BRDK_UPDATE_NO_ID_MATCH := 1, (*Configuration ID of the update and machine does not match.*)
		BRDK_UPDATE_VERSION_ERROR_FORMAT := 2, (*Format of the version does not comply with x.x.x.*)
		BRDK_UPDATE_VERSIONS_EQUAL := 3, (*Same version on the update package and the machine.*)
		BRDK_UPDATE_VERSION_NEW_SMALLER := 4, (*Update version smaller than machine version.*)
		BRDK_UPDATE_VERSION_NEW_GREATER := 5 (*Update version greater than machine version.*)
		);
	brdk_update_manager_upd_loc_typ :
		( (*Location of the update package.*)
		BRDK_UPDATE_LOCATION_USER := 0, (*Update package can both be located on USER partition only.*)
		BRDK_UPDATE_LOCATION_USB := 1 (*Update package can both be located on USB only.*)
		) := BRDK_UPDATE_LOCATION_USER;
	brdk_update_manager_cmd_typ : 	STRUCT  (*Commands.*)
		checkForUpdate : BOOL := FALSE; (*Checks for an update.*)
		update : BOOL := FALSE; (*Update PLC.*)
		updateReboot : BOOL := FALSE; (*Update PLC and rebootPLC afterwards.*)
		deleteUpdate : BOOL := FALSE; (*Deletes an update.*)
		errorReset : BOOL := FALSE; (*Resets errors.*)
	END_STRUCT;
	brdk_update_dist_ftp_int_typ : 	STRUCT  (*Distribute internal variables.*)
		state : DINT := 0; (*Internal state.*)
		DevLink_0 : DevLink; (*DevLink.*)
		DevUnlink_0 : DevUnlink; (*DevUnlink.*)
		FileCopy_0 : FileCopy; (*FileCopy.*)
		DirCopy_0 : DirCopy; (*DirCopy.*)
		cIdx : USINT := 0; (*Client idx.*)
		paramStr : STRING[200] := ''; (*Parameter string.*)
		brdkUpdateCheck_0 : brdkUpdateCheck; (*brdkUpdateCheck.*)
		brdkUpdateDelete_0 : brdkUpdateDelete; (*brdkUpdateDelete.*)
	END_STRUCT;
	brdk_update_dist_ftp_client_typ : 	STRUCT  (*PLC client structure.*)
		pIPAddress : UDINT := 0; (*String pointer to IP address of the PLC client.*)
		pUser : UDINT := 0; (*String pointer to FTP user name.*)
		pPassword : UDINT := 0; (*String pointer to FTP password.*)
	END_STRUCT;
	brdk_update_dist_ftp_cmd_typ : 	STRUCT  (*Command structure.*)
		distributeUpdate : BOOL := FALSE; (*Distributes the update to the clients in the client list.*)
		checkUpdate : BOOL := FALSE; (*Reads the data from the update.*)
		deleteUpdate : BOOL := FALSE; (*Deletes an update.*)
		errorReset : BOOL := FALSE; (*Resets errors.*)
	END_STRUCT;
	brdk_update_check_internal_typ : 	STRUCT  (*Read internal variables.*)
		state : DINT := 0; (*Internal state.*)
		brdkFileRead_0 : brdkFileRead; (*brdkFileRead.*)
		buffer : ARRAY[0..1999]OF USINT; (*Read buffer.*)
		simulation : BOOL := FALSE; (*Simulation active.*)
		ArProjectGetPackageInfo_0 : ArProjectGetPackageInfo; (*ArProjectGetPackageInfo.*)
		position : DINT; (*Find position.*)
		FileInfo_0 : FileInfo; (*Read update file info*)
		updateFileInfo : fiFILE_INFO; (*File info structure*)
	END_STRUCT;
	brdk_update_delete_internal_typ : 	STRUCT  (*Delete internal variables.*)
		state : DINT := 0; (*Internal state.*)
		brdkUpdateCheck_0 : brdkUpdateCheck; (*brdkUpdateCheck.*)
		FileDelete_0 : FileDelete; (*FileDelete.*)
		DirDeleteEx_0 : DirDeleteEx; (*DirDeleteEx.*)
	END_STRUCT;
END_TYPE
```

#### brdkUpdate.var - Exported constants
```iecst
VAR CONSTANT
	BRDK_UPDATE_USER_FILE_DEVICE : STRING[80] := 'BRDK_UPDATE_USER'; (*USER partition file device name.*)
	BRDK_UPDATE_USB_FILE_DEVICE : STRING[80] := 'BRDK_UPDATE_USB'; (*USB file device name.*)
	BRDK_UPDATE_USER_PATH : STRING[80] := 'F:\'; (*Path for USER partition.*)
	BRDK_UPDATE_DEFAULT_FILE_NAME : STRING[80] := 'arnbcfg.xml'; (*Default file name for update xml file.*)
	BRDK_UPDATE_AR_TRANSFER_PATH : STRING[80] := '\artransfer.br'; (*Default path from update folder to 'artransfer.br' file.*)
	BRDK_UPDATE_MAX_VERSION_NUM_LEN : USINT := 10; (*Max length of each verion number string.*)
	BRDK_UPDATE_PIP_FILE_ERROR : DINT := -535835272; (*Wrong format in arnbcfg.xml file.*)
	BRDK_UPDATE_POINTER_ERROR : DINT := -535835273; (*Pointer error.*)
	BRDK_UPDATE_FORMAT_ERROR : DINT := -535835274; (*Format error.*)
	BRDK_UPDATE_MAX_FTP_CLIENTS : USINT := 2; (*Max. number of FTP clients in the list.*)
	BRDK_UPDATE_FTP_DEVICE_NAME : STRING[80] := 'BRDK_UPDATE_FTP'; (*FTP device name.*)
END_VAR
```
